LIN {X 0,Y 247.203,Z 467.136,A -85,B 0,C 180,E1 -18801.825,E2 -18801.825} C_VEL
LIN {X 0,Y 246.923,Z 469.012,A -85,B 0,C 180,E1 -18805.099,E2 -18805.099} C_VEL
LIN {X 0,Y 246.987,Z 469.369,A -85,B 0,C 180,E1 -18806.735,E2 -18806.735} C_VEL
LIN {X 0,Y 247.048,Z 469.339,A -85,B 0,C 180,E1 -18808.367,E2 -18808.367} C_VEL
LIN {X 0,Y 247.097,Z 468.891,A -85,B 0,C 180,E1 -18809.997,E2 -18809.997} C_VEL
LIN {X 0,Y 247.079,Z 468.012,A -85,B 0,C 180,E1 -18811.627,E2 -18811.627} C_VEL
LIN {X 0,Y 247.04,Z 466.727,A -85,B 0,C 180,E1 -18813.258,E2 -18813.258} C_VEL
LIN {X 0,Y 247.021,Z 464.571,A -85,B 0,C 180,E1 -18815.261,E2 -18815.261} C_VEL
LIN {X 0,Y 247.246,Z 460.184,A -85,B 0,C 180,E1 -18818.167,E2 -18818.167} C_VEL
LIN {X 0,Y 247.68,Z 455.238,A -85,B 0,C 180,E1 -18820.624,E2 -18820.624} C_VEL
LIN {X 0,Y 248.441,Z 448.994,A -85,B 0,C 180,E1 -18823.075,E2 -18823.075} C_VEL
LIN {X 0,Y 249.662,Z 441.211,A -85,B 0,C 180,E1 -18825.506,E2 -18825.506} C_VEL
LIN {X 0,Y 250.752,Z 434.213,A -85,B 0,C 180,E1 -18827.293,E2 -18827.293} C_VEL
LIN {X 0,Y 252.36,Z 424.659,A -85,B 0,C 180,E1 -18829.286,E2 -18829.286} C_VEL
LIN {X 0,Y 253.976,Z 413.923,A -85,B 0,C 180,E1 -18831.079,E2 -18831.079} C_VEL
LIN {X 0,Y 255.738,Z 402.097,A -85,B 0,C 180,E1 -18832.622,E2 -18832.622} C_VEL
LIN {X 0,Y 257.174,Z 390.548,A -85,B 0,C 180,E1 -18833.765,E2 -18833.765} C_VEL
LIN {X 0,Y 258.492,Z 377.529,A -85,B 0,C 180,E1 -18834.704,E2 -18834.704} C_VEL
LIN {X 0,Y 259.341,Z 364.879,A -85,B 0,C 180,E1 -18835.313,E2 -18835.313} C_VEL
LIN {X 0,Y 260.976,Z 308.011,A -85,B 0,C 180,E1 -18836.87,E2 -18836.87} C_VEL
LIN {X 0,Y 256.67,Z 271.586,A -85,B 0,C 180,E1 -18838.358,E2 -18838.358} C_VEL
LIN {X 0,Y 255.368,Z 263.288,A -85,B 0,C 180,E1 -18838.738,E2 -18838.738} C_VEL
LIN {X 0,Y 252.839,Z 256.196,A -85,B 0,C 180,E1 -18839.225,E2 -18839.225} C_VEL
LIN {X 0,Y 250.431,Z 244.513,A -85,B 0,C 180,E1 -18843.344,E2 -18843.344} C_VEL
LIN {X 0,Y 249.071,Z 238.465,A -85,B 0,C 180,E1 -18845.637,E2 -18845.637} C_VEL
LIN {X 0,Y 249.01,Z 238.469,A -85,B 0,C 180,E1 -18848.375,E2 -18848.375} C_VEL
LIN {X 0,Y 248.991,Z 238.469,A -85,B 0,C 180,E1 -18852.788,E2 -18852.788} C_VEL
LIN {X 0,Y 249.034,Z 238.465,A -85,B 0,C 180,E1 -18857.367,E2 -18857.367} C_VEL
LIN {X 0,Y 249.022,Z 238.468,A -85,B 0,C 180,E1 -18861.619,E2 -18861.619} C_VEL
LIN {X 0,Y 249.017,Z 238.467,A -85,B 0,C 180,E1 -18865.635,E2 -18865.635} C_VEL
LIN {X 0,Y 249.021,Z 238.466,A -85,B 0,C 180,E1 -18869.469,E2 -18869.469} C_VEL
LIN {X 0,Y 249.044,Z 238.463,A -85,B 0,C 180,E1 -18873.159,E2 -18873.159} C_VEL
LIN {X 0,Y 249.081,Z 238.456,A -85,B 0,C 180,E1 -18876.733,E2 -18876.733} C_VEL
LIN {X 0,Y 249.112,Z 238.452,A -85,B 0,C 180,E1 -18880.212,E2 -18880.212} C_VEL
LIN {X 0,Y 249.161,Z 238.449,A -85,B 0,C 180,E1 -18883.617,E2 -18883.617} C_VEL
LIN {X 0,Y 249.205,Z 238.44,A -85,B 0,C 180,E1 -18888.614,E2 -18888.614} C_VEL
LIN {X 0,Y 249.42,Z 238.411,A -85,B 0,C 180,E1 -18891.901,E2 -18891.901} C_VEL
LIN {X 0,Y 249.257,Z 238.437,A -85,B 0,C 180,E1 -18895.148,E2 -18895.148} C_VEL
LIN {X 0,Y 249.634,Z 238.385,A -85,B 0,C 180,E1 -18898.387,E2 -18898.387} C_VEL
LIN {X 0,Y 249.631,Z 238.366,A -85,B 0,C 180,E1 -18901.613,E2 -18901.613} C_VEL
LIN {X 0,Y 249.393,Z 238.414,A -85,B 0,C 180,E1 -18906.767,E2 -18906.767} C_VEL
LIN {X 0,Y 249.297,Z 238.427,A -85,B 0,C 180,E1 -18909.738,E2 -18909.738} C_VEL
LIN {X 0,Y 249.132,Z 238.432,A -85,B 0,C 180,E1 -18914.708,E2 -18914.708} C_VEL
LIN {X 0,Y 249.058,Z 238.455,A -85,B 0,C 180,E1 -18918.084,E2 -18918.084} C_VEL
LIN {X 0,Y 249.012,Z 238.464,A -85,B 0,C 180,E1 -18921.525,E2 -18921.525} C_VEL
LIN {X 0,Y 249.084,Z 238.456,A -85,B 0,C 180,E1 -18925.478,E2 -18925.478} C_VEL
LIN {X 0,Y 249.042,Z 238.46,A -85,B 0,C 180,E1 -18928.992,E2 -18928.992} C_VEL
LIN {X 0,Y 249.002,Z 238.469,A -85,B 0,C 180,E1 -18932.43,E2 -18932.43} C_VEL
LIN {X 0,Y 249.035,Z 238.465,A -85,B 0,C 180,E1 -18936.345,E2 -18936.345} C_VEL
LIN {X 0,Y 249.053,Z 238.461,A -85,B 0,C 180,E1 -18940.469,E2 -18940.469} C_VEL
LIN {X 0,Y 248.992,Z 238.457,A -85,B 0,C 180,E1 -18944.882,E2 -18944.882} C_VEL
LIN {X 0,Y 248.999,Z 238.46,A -85,B 0,C 180,E1 -18947.368,E2 -18947.368} C_VEL
LIN {X 0,Y 249.026,Z 238.457,A -85,B 0,C 180,E1 -18952.206,E2 -18952.206} C_VEL
LIN {X 0,Y 249.03,Z 238.464,A -85,B 0,C 180,E1 -18955.645,E2 -18955.645} C_VEL
LIN {X 0,Y 249.036,Z 238.464,A -85,B 0,C 180,E1 -18959.478,E2 -18959.478} C_VEL
LIN {X 0,Y 249.059,Z 238.459,A -85,B 0,C 180,E1 -18963.167,E2 -18963.167} C_VEL
LIN {X 0,Y 249.053,Z 238.458,A -85,B 0,C 180,E1 -18966.736,E2 -18966.736} C_VEL
LIN {X 0,Y 249.116,Z 238.454,A -85,B 0,C 180,E1 -18971.159,E2 -18971.159} C_VEL
LIN {X 0,Y 249.116,Z 238.559,A -85,B 0,C 180,E1 -18971.564,E2 -18971.564} C_VEL
LIN {X 0,Y 250.194,Z 241.443,A -85,B 0,C 180,E1 -18971.772,E2 -18971.772} C_VEL
LIN {X 0,Y 256.891,Z 255.902,A -85,B 0,C 180,E1 -18972.914,E2 -18972.914} C_VEL
LIN {X 0,Y 262.003,Z 270.873,A -85,B 0,C 180,E1 -18973.855,E2 -18973.855} C_VEL
LIN {X 0,Y 259.67,Z 343.56,A -85,B 0,C 180,E1 -18975.827,E2 -18975.827} C_VEL
LIN {X 0,Y 258.82,Z 356.25,A -85,B 0,C 180,E1 -18976.46,E2 -18976.46} C_VEL
LIN {X 0,Y 257.913,Z 367.725,A -85,B 0,C 180,E1 -18977.313,E2 -18977.313} C_VEL
LIN {X 0,Y 256.76,Z 380.047,A -85,B 0,C 180,E1 -18978.558,E2 -18978.558} C_VEL
LIN {X 0,Y 255.064,Z 391.695,A -85,B 0,C 180,E1 -18980.088,E2 -18980.088} C_VEL
LIN {X 0,Y 253.487,Z 402.134,A -85,B 0,C 180,E1 -18981.835,E2 -18981.835} C_VEL
LIN {X 0,Y 252.061,Z 410.678,A -85,B 0,C 180,E1 -18983.6,E2 -18983.6} C_VEL
LIN {X 0,Y 250.811,Z 418.54,A -85,B 0,C 180,E1 -18985.584,E2 -18985.584} C_VEL
LIN {X 0,Y 249.419,Z 426.253,A -85,B 0,C 180,E1 -18987.985,E2 -18987.985} C_VEL
LIN {X 0,Y 248.629,Z 431.513,A -85,B 0,C 180,E1 -18990.003,E2 -18990.003} C_VEL
LIN {X 0,Y 247.945,Z 436.619,A -85,B 0,C 180,E1 -18992.44,E2 -18992.44} C_VEL
LIN {X 0,Y 247.504,Z 440.592,A -85,B 0,C 180,E1 -18994.889,E2 -18994.889} C_VEL
LIN {X 0,Y 247.252,Z 442.647,A -85,B 0,C 180,E1 -18996.531,E2 -18996.531} C_VEL
LIN {X 0,Y 247.006,Z 444.293,A -85,B 0,C 180,E1 -18998.181,E2 -18998.181} C_VEL
LIN {X 0,Y 246.9,Z 445.534,A -85,B 0,C 180,E1 -18999.836,E2 -18999.836} C_VEL
LIN {X 0,Y 246.89,Z 446.331,A -85,B 0,C 180,E1 -19001.496,E2 -19001.496} C_VEL
LIN {X 0,Y 247.048,Z 446.719,A -85,B 0,C 180,E1 -19003.157,E2 -19003.157} C_VEL
LIN {X 0,Y 247.277,Z 446.714,A -85,B 0,C 180,E1 -19004.908,E2 -19004.908} C_VEL
LIN {X 0,Y 247.511,Z 446.329,A -85,B 0,C 180,E1 -19006.497,E2 -19006.497} C_VEL
LIN {X 0,Y 247.958,Z 445.48,A -85,B 0,C 180,E1 -19008.168,E2 -19008.168} C_VEL
LIN {X 0,Y 248.534,Z 444.221,A -85,B 0,C 180,E1 -19009.838,E2 -19009.838} C_VEL
LIN {X 0,Y 249.653,Z 441.509,A -85,B 0,C 180,E1 -19012.337,E2 -19012.337} C_VEL
LIN {X 0,Y 251.127,Z 437.727,A -85,B 0,C 180,E1 -19014.822,E2 -19014.822} C_VEL
LIN {X 0,Y 253.115,Z 432.322,A -85,B 0,C 180,E1 -19017.48,E2 -19017.48} C_VEL
LIN {X 0,Y 255.623,Z 425.225,A -85,B 0,C 180,E1 -19020.117,E2 -19020.117} C_VEL
LIN {X 0,Y 258.288,Z 417.007,A -85,B 0,C 180,E1 -19022.487,E2 -19022.487} C_VEL
LIN {X 0,Y 260.828,Z 408.416,A -85,B 0,C 180,E1 -19024.461,E2 -19024.461} C_VEL
LIN {X 0,Y 263.568,Z 398.096,A -85,B 0,C 180,E1 -19026.333,E2 -19026.333} C_VEL
LIN {X 0,Y 266.096,Z 387.21,A -85,B 0,C 180,E1 -19027.883,E2 -19027.883} C_VEL
LIN {X 0,Y 268.227,Z 375.469,A -85,B 0,C 180,E1 -19029.205,E2 -19029.205} C_VEL
LIN {X 0,Y 270.041,Z 363.177,A -85,B 0,C 180,E1 -19030.222,E2 -19030.222} C_VEL
LIN {X 0,Y 271.458,Z 349.994,A -85,B 0,C 180,E1 -19030.986,E2 -19030.986} C_VEL
LIN {X 0,Y 272.232,Z 337.682,A -85,B 0,C 180,E1 -19031.434,E2 -19031.434} C_VEL
LIN {X 0,Y 274.351,Z 284.179,A -85,B 0,C 180,E1 -19032.822,E2 -19032.822} C_VEL
LIN {X 0,Y 267.59,Z 269.785,A -85,B 0,C 180,E1 -19034.382,E2 -19034.382} C_VEL
LIN {X 0,Y 261.114,Z 257.839,A -85,B 0,C 180,E1 -19035.925,E2 -19035.925} C_VEL
LIN {X 0,Y 253.708,Z 246.432,A -85,B 0,C 180,E1 -19037.752,E2 -19037.752} C_VEL
LIN {X 0,Y 251.454,Z 242.928,A -85,B 0,C 180,E1 -19038.342,E2 -19038.342} C_VEL
LIN {X 0,Y 249.713,Z 240.612,A -85,B 0,C 180,E1 -19038.795,E2 -19038.795} C_VEL
LIN {X 0,Y 249.083,Z 238.458,A -85,B 0,C 180,E1 -19039.037,E2 -19039.037} C_VEL
LIN {X 0,Y 249.052,Z 238.46,A -85,B 0,C 180,E1 -19043.658,E2 -19043.658} C_VEL
LIN {X 0,Y 249.031,Z 238.463,A -85,B 0,C 180,E1 -19047.845,E2 -19047.845} C_VEL
LIN {X 0,Y 249.089,Z 238.456,A -85,B 0,C 180,E1 -19051.337,E2 -19051.337} C_VEL
LIN {X 0,Y 249.125,Z 238.452,A -85,B 0,C 180,E1 -19054.965,E2 -19054.965} C_VEL
LIN {X 0,Y 249.08,Z 238.458,A -85,B 0,C 180,E1 -19058.604,E2 -19058.604} C_VEL
LIN {X 0,Y 249.187,Z 238.438,A -85,B 0,C 180,E1 -19063.618,E2 -19063.618} C_VEL
LIN {X 0,Y 249.212,Z 238.432,A -85,B 0,C 180,E1 -19068.614,E2 -19068.614} C_VEL
LIN {X 0,Y 249.434,Z 238.413,A -85,B 0,C 180,E1 -19071.901,E2 -19071.901} C_VEL
LIN {X 0,Y 249.271,Z 238.431,A -85,B 0,C 180,E1 -19075.148,E2 -19075.148} C_VEL
LIN {X 0,Y 249.657,Z 238.373,A -85,B 0,C 180,E1 -19078.387,E2 -19078.387} C_VEL
LIN {X 0,Y 249.651,Z 238.383,A -85,B 0,C 180,E1 -19081.613,E2 -19081.613} C_VEL
LIN {X 0,Y 249.332,Z 238.415,A -85,B 0,C 180,E1 -19083.677,E2 -19083.677} C_VEL
LIN {X 0,Y 248.579,Z 238.52,A -85,B 0,C 180,E1 -19085.027,E2 -19085.027} C_VEL
LIN {X 0,Y 245.722,Z 238.875,A -85,B 0,C 180,E1 -19087.229,E2 -19087.229} C_VEL
LIN {X 0,Y 243.329,Z 239.172,A -85,B 0,C 180,E1 -19089.022,E2 -19089.022} C_VEL
LIN {X 0,Y 242.275,Z 239.305,A -85,B 0,C 180,E1 -19090.411,E2 -19090.411} C_VEL
LIN {X 0,Y 242.171,Z 239.31,A -85,B 0,C 180,E1 -19090.882,E2 -19090.882} C_VEL
LIN {X 0,Y 242.108,Z 239.325,A -85,B 0,C 180,E1 -19095.144,E2 -19095.144} C_VEL
LIN {X 0,Y 242.018,Z 239.335,A -85,B 0,C 180,E1 -19098.628,E2 -19098.628} C_VEL
LIN {X 0,Y 241.963,Z 239.336,A -85,B 0,C 180,E1 -19102.185,E2 -19102.185} C_VEL
LIN {X 0,Y 241.978,Z 239.332,A -85,B 0,C 180,E1 -19105.827,E2 -19105.827} C_VEL
LIN {X 0,Y 241.953,Z 239.336,A -85,B 0,C 180,E1 -19109.59,E2 -19109.59} C_VEL
LIN {X 0,Y 241.96,Z 239.335,A -85,B 0,C 180,E1 -19113.496,E2 -19113.496} C_VEL
LIN {X 0,Y 241.978,Z 239.314,A -85,B 0,C 180,E1 -19117.584,E2 -19117.584} C_VEL
LIN {X 0,Y 241.923,Z 239.349,A -85,B 0,C 180,E1 -19121.926,E2 -19121.926} C_VEL
LIN {X 0,Y 241.904,Z 239.396,A -85,B 0,C 180,E1 -19124.093,E2 -19124.093} C_VEL
LIN {X 0,Y 244.427,Z 247.713,A -85,B 0,C 180,E1 -19128.381,E2 -19128.381} C_VEL
LIN {X 0,Y 246.312,Z 254.372,A -85,B 0,C 180,E1 -19131.43,E2 -19131.43} C_VEL
LIN {X 0,Y 248.91,Z 258.983,A -85,B 0,C 180,E1 -19132.159,E2 -19132.159} C_VEL
LIN {X 0,Y 254.848,Z 270.286,A -85,B 0,C 180,E1 -19133.768,E2 -19133.768} C_VEL
LIN {X 0,Y 261.821,Z 284.82,A -85,B 0,C 180,E1 -19135.559,E2 -19135.559} C_VEL
LIN {X 0,Y 263.955,Z 290.021,A -85,B 0,C 180,E1 -19136.105,E2 -19136.105} C_VEL
LIN {X 0,Y 267.543,Z 313.214,A -85,B 0,C 180,E1 -19137.473,E2 -19137.473} C_VEL
LIN {X 0,Y 265.351,Z 364.24,A -85,B 0,C 180,E1 -19138.851,E2 -19138.851} C_VEL
LIN {X 0,Y 263.985,Z 377.838,A -85,B 0,C 180,E1 -19139.486,E2 -19139.486} C_VEL
LIN {X 0,Y 261.967,Z 390.55,A -85,B 0,C 180,E1 -19140.354,E2 -19140.354} C_VEL
LIN {X 0,Y 259.554,Z 402.464,A -85,B 0,C 180,E1 -19141.495,E2 -19141.495} C_VEL
LIN {X 0,Y 256.853,Z 413.883,A -85,B 0,C 180,E1 -19142.942,E2 -19142.942} C_VEL
LIN {X 0,Y 253.958,Z 424.203,A -85,B 0,C 180,E1 -19144.599,E2 -19144.599} C_VEL
LIN {X 0,Y 251.143,Z 433.502,A -85,B 0,C 180,E1 -19146.498,E2 -19146.498} C_VEL
LIN {X 0,Y 248.11,Z 442.53,A -85,B 0,C 180,E1 -19148.828,E2 -19148.828} C_VEL
LIN {X 0,Y 245.748,Z 449.9,A -85,B 0,C 180,E1 -19151.258,E2 -19151.258} C_VEL
LIN {X 0,Y 243.418,Z 456.556,A -85,B 0,C 180,E1 -19154.079,E2 -19154.079} C_VEL
LIN {X 0,Y 241.79,Z 461.028,A -85,B 0,C 180,E1 -19156.552,E2 -19156.552} C_VEL
LIN {X 0,Y 241.123,Z 463.407,A -85,B 0,C 180,E1 -19158.225,E2 -19158.225} C_VEL
LIN {X 0,Y 240.555,Z 465.363,A -85,B 0,C 180,E1 -19159.902,E2 -19159.902} C_VEL
LIN {X 0,Y 240.162,Z 466.905,A -85,B 0,C 180,E1 -19161.584,E2 -19161.584} C_VEL
LIN {X 0,Y 239.847,Z 468.719,A -85,B 0,C 180,E1 -19164.954,E2 -19164.954} C_VEL
LIN {X 0,Y 239.882,Z 469.052,A -85,B 0,C 180,E1 -19166.638,E2 -19166.638} C_VEL
LIN {X 0,Y 239.975,Z 468.998,A -85,B 0,C 180,E1 -19168.319,E2 -19168.319} C_VEL
LIN {X 0,Y 240.022,Z 468.506,A -85,B 0,C 180,E1 -19169.997,E2 -19169.997} C_VEL
LIN {X 0,Y 240.006,Z 467.602,A -85,B 0,C 180,E1 -19171.675,E2 -19171.675} C_VEL
LIN {X 0,Y 239.955,Z 466.293,A -85,B 0,C 180,E1 -19173.355,E2 -19173.355} C_VEL
LIN {X 0,Y 239.95,Z 464.329,A -85,B 0,C 180,E1 -19175.226,E2 -19175.226} C_VEL
LIN {X 0,Y 240.105,Z 461.075,A -85,B 0,C 180,E1 -19177.565,E2 -19177.565} C_VEL
LIN {X 0,Y 240.463,Z 456.468,A -85,B 0,C 180,E1 -19180.096,E2 -19180.096} C_VEL
LIN {X 0,Y 241.321,Z 449.467,A -85,B 0,C 180,E1 -19183.04,E2 -19183.04} C_VEL
LIN {X 0,Y 242.562,Z 441.881,A -85,B 0,C 180,E1 -19185.541,E2 -19185.541} C_VEL
LIN {X 0,Y 243.714,Z 434.867,A -85,B 0,C 180,E1 -19187.425,E2 -19187.425} C_VEL
LIN {X 0,Y 245.28,Z 425.71,A -85,B 0,C 180,E1 -19189.451,E2 -19189.451} C_VEL
LIN {X 0,Y 246.938,Z 415.436,A -85,B 0,C 180,E1 -19191.271,E2 -19191.271} C_VEL
LIN {X 0,Y 248.456,Z 405.625,A -85,B 0,C 180,E1 -19192.663,E2 -19192.663} C_VEL
LIN {X 0,Y 250.176,Z 393.195,A -85,B 0,C 180,E1 -19194.032,E2 -19194.032} C_VEL
LIN {X 0,Y 251.486,Z 381.401,A -85,B 0,C 180,E1 -19194.998,E2 -19194.998} C_VEL
LIN {X 0,Y 252.523,Z 368.688,A -85,B 0,C 180,E1 -19195.715,E2 -19195.715} C_VEL
LIN {X 0,Y 253.145,Z 352.376,A -85,B 0,C 180,E1 -19196.255,E2 -19196.255} C_VEL
LIN {X 0,Y 254.295,Z 307.444,A -85,B 0,C 180,E1 -19197.504,E2 -19197.504} C_VEL
LIN {X 0,Y 249.978,Z 270.919,A -85,B 0,C 180,E1 -19199.053,E2 -19199.053} C_VEL
LIN {X 0,Y 248.956,Z 265.195,A -85,B 0,C 180,E1 -19199.339,E2 -19199.339} C_VEL
LIN {X 0,Y 245.586,Z 255.846,A -85,B 0,C 180,E1 -19200.008,E2 -19200.008} C_VEL
LIN {X 0,Y 243.121,Z 244.14,A -85,B 0,C 180,E1 -19204.303,E2 -19204.303} C_VEL
LIN {X 0,Y 242.004,Z 239.343,A -85,B 0,C 180,E1 -19206.205,E2 -19206.205} C_VEL
LIN {X 0,Y 241.939,Z 239.35,A -85,B 0,C 180,E1 -19209.714,E2 -19209.714} C_VEL
LIN {X 0,Y 241.916,Z 239.351,A -85,B 0,C 180,E1 -19214.196,E2 -19214.196} C_VEL
LIN {X 0,Y 241.958,Z 239.347,A -85,B 0,C 180,E1 -19218.082,E2 -19218.082} C_VEL
LIN {X 0,Y 241.978,Z 239.342,A -85,B 0,C 180,E1 -19222.416,E2 -19222.416} C_VEL
LIN {X 0,Y 241.953,Z 239.344,A -85,B 0,C 180,E1 -19226.503,E2 -19226.503} C_VEL
LIN {X 0,Y 242.007,Z 239.338,A -85,B 0,C 180,E1 -19230.584,E2 -19230.584} C_VEL
LIN {X 0,Y 242.037,Z 239.334,A -85,B 0,C 180,E1 -19234.18,E2 -19234.18} C_VEL
LIN {X 0,Y 242.056,Z 239.331,A -85,B 0,C 180,E1 -19238.273,E2 -19238.273} C_VEL
LIN {X 0,Y 242.121,Z 239.326,A -85,B 0,C 180,E1 -19243.283,E2 -19243.283} C_VEL
LIN {X 0,Y 242.141,Z 239.32,A -85,B 0,C 180,E1 -19248.278,E2 -19248.278} C_VEL
LIN {X 0,Y 242.366,Z 239.29,A -85,B 0,C 180,E1 -19251.664,E2 -19251.664} C_VEL
LIN {X 0,Y 242.218,Z 239.313,A -85,B 0,C 180,E1 -19255.006,E2 -19255.006} C_VEL
LIN {X 0,Y 242.595,Z 239.261,A -85,B 0,C 180,E1 -19258.34,E2 -19258.34} C_VEL
LIN {X 0,Y 242.592,Z 239.241,A -85,B 0,C 180,E1 -19261.66,E2 -19261.66} C_VEL
LIN {X 0,Y 242.372,Z 239.29,A -85,B 0,C 180,E1 -19266.74,E2 -19266.74} C_VEL
LIN {X 0,Y 242.226,Z 239.308,A -85,B 0,C 180,E1 -19270.026,E2 -19270.026} C_VEL
LIN {X 0,Y 242.083,Z 239.311,A -85,B 0,C 180,E1 -19275.146,E2 -19275.146} C_VEL
LIN {X 0,Y 241.995,Z 239.338,A -85,B 0,C 180,E1 -19278.631,E2 -19278.631} C_VEL
LIN {X 0,Y 241.955,Z 239.344,A -85,B 0,C 180,E1 -19282.186,E2 -19282.186} C_VEL
LIN {X 0,Y 242.037,Z 239.334,A -85,B 0,C 180,E1 -19285.842,E2 -19285.842} C_VEL
LIN {X 0,Y 241.978,Z 239.338,A -85,B 0,C 180,E1 -19289.588,E2 -19289.588} C_VEL
LIN {X 0,Y 241.954,Z 239.342,A -85,B 0,C 180,E1 -19293.497,E2 -19293.497} C_VEL
LIN {X 0,Y 241.982,Z 239.341,A -85,B 0,C 180,E1 -19297.584,E2 -19297.584} C_VEL
LIN {X 0,Y 241.959,Z 239.344,A -85,B 0,C 180,E1 -19301.918,E2 -19301.918} C_VEL
LIN {X 0,Y 241.917,Z 239.336,A -85,B 0,C 180,E1 -19305.804,E2 -19305.804} C_VEL
LIN {X 0,Y 241.93,Z 239.347,A -85,B 0,C 180,E1 -19310.284,E2 -19310.284} C_VEL
LIN {X 0,Y 241.966,Z 239.342,A -85,B 0,C 180,E1 -19314.494,E2 -19314.494} C_VEL
LIN {X 0,Y 241.961,Z 239.345,A -85,B 0,C 180,E1 -19318.485,E2 -19318.485} C_VEL
LIN {X 0,Y 241.991,Z 239.341,A -85,B 0,C 180,E1 -19322.317,E2 -19322.317} C_VEL
LIN {X 0,Y 242.033,Z 239.335,A -85,B 0,C 180,E1 -19326.019,E2 -19326.019} C_VEL
LIN {X 0,Y 242.052,Z 239.333,A -85,B 0,C 180,E1 -19330.775,E2 -19330.775} C_VEL
LIN {X 0,Y 243.117,Z 242.269,A -85,B 0,C 180,E1 -19331.011,E2 -19331.011} C_VEL
LIN {X 0,Y 250.739,Z 258.529,A -85,B 0,C 180,E1 -19332.364,E2 -19332.364} C_VEL
LIN {X 0,Y 255.469,Z 272.48,A -85,B 0,C 180,E1 -19333.274,E2 -19333.274} C_VEL
LIN {X 0,Y 253.06,Z 343.957,A -85,B 0,C 180,E1 -19335.258,E2 -19335.258} C_VEL
LIN {X 0,Y 252.18,Z 356.417,A -85,B 0,C 180,E1 -19335.89,E2 -19335.89} C_VEL
LIN {X 0,Y 251.252,Z 367.929,A -85,B 0,C 180,E1 -19336.765,E2 -19336.765} C_VEL
LIN {X 0,Y 250.056,Z 380.285,A -85,B 0,C 180,E1 -19338.041,E2 -19338.041} C_VEL
LIN {X 0,Y 248.302,Z 391.953,A -85,B 0,C 180,E1 -19339.609,E2 -19339.609} C_VEL
LIN {X 0,Y 246.664,Z 402.405,A -85,B 0,C 180,E1 -19341.401,E2 -19341.401} C_VEL
LIN {X 0,Y 245.039,Z 411.836,A -85,B 0,C 180,E1 -19343.416,E2 -19343.416} C_VEL
LIN {X 0,Y 243.514,Z 420.897,A -85,B 0,C 180,E1 -19345.866,E2 -19345.866} C_VEL
LIN {X 0,Y 242.144,Z 428.227,A -85,B 0,C 180,E1 -19348.34,E2 -19348.34} C_VEL
LIN {X 0,Y 241.301,Z 434.084,A -85,B 0,C 180,E1 -19350.837,E2 -19350.837} C_VEL
LIN {X 0,Y 240.613,Z 438.721,A -85,B 0,C 180,E1 -19353.352,E2 -19353.352} C_VEL
LIN {X 0,Y 240.256,Z 442.364,A -85,B 0,C 180,E1 -19355.967,E2 -19355.967} C_VEL
LIN {X 0,Y 239.883,Z 444.8,A -85,B 0,C 180,E1 -19358.426,E2 -19358.426} C_VEL
LIN {X 0,Y 239.808,Z 445.979,A -85,B 0,C 180,E1 -19360.13,E2 -19360.13} C_VEL
LIN {X 0,Y 239.99,Z 447.071,A -85,B 0,C 180,E1 -19363.551,E2 -19363.551} C_VEL
LIN {X 0,Y 240.239,Z 447.035,A -85,B 0,C 180,E1 -19365.267,E2 -19365.267} C_VEL
LIN {X 0,Y 240.544,Z 446.572,A -85,B 0,C 180,E1 -19366.99,E2 -19366.99} C_VEL
LIN {X 0,Y 241.021,Z 445.678,A -85,B 0,C 180,E1 -19368.71,E2 -19368.71} C_VEL
LIN {X 0,Y 242.296,Z 442.972,A -85,B 0,C 180,E1 -19371.845,E2 -19371.845} C_VEL
LIN {X 0,Y 243.926,Z 439.154,A -85,B 0,C 180,E1 -19374.695,E2 -19374.695} C_VEL
LIN {X 0,Y 246.135,Z 433.406,A -85,B 0,C 180,E1 -19377.728,E2 -19377.728} C_VEL
LIN {X 0,Y 248.43,Z 427.372,A -85,B 0,C 180,E1 -19380.142,E2 -19380.142} C_VEL
LIN {X 0,Y 251.163,Z 419.752,A -85,B 0,C 180,E1 -19382.54,E2 -19382.54} C_VEL
LIN {X 0,Y 253.726,Z 411.531,A -85,B 0,C 180,E1 -19384.599,E2 -19384.599} C_VEL
LIN {X 0,Y 256.552,Z 401.625,A -85,B 0,C 180,E1 -19386.571,E2 -19386.571} C_VEL
LIN {X 0,Y 259.479,Z 390.344,A -85,B 0,C 180,E1 -19388.319,E2 -19388.319} C_VEL
LIN {X 0,Y 261.603,Z 379.544,A -85,B 0,C 180,E1 -19389.645,E2 -19389.645} C_VEL
LIN {X 0,Y 263.426,Z 368.513,A -85,B 0,C 180,E1 -19390.69,E2 -19390.69} C_VEL
LIN {X 0,Y 265.152,Z 355.149,A -85,B 0,C 180,E1 -19391.604,E2 -19391.604} C_VEL
LIN {X 0,Y 266.232,Z 341.893,A -85,B 0,C 180,E1 -19392.182,E2 -19392.182} C_VEL
LIN {X 0,Y 268.615,Z 286.422,A -85,B 0,C 180,E1 -19393.657,E2 -19393.657} C_VEL
LIN {X 0,Y 261.963,Z 272.273,A -85,B 0,C 180,E1 -19395.267,E2 -19395.267} C_VEL
LIN {X 0,Y 256.197,Z 261.74,A -85,B 0,C 180,E1 -19396.701,E2 -19396.701} C_VEL
LIN {X 0,Y 247.39,Z 248.085,A -85,B 0,C 180,E1 -19398.999,E2 -19398.999} C_VEL
LIN {X 0,Y 245.215,Z 244.854,A -85,B 0,C 180,E1 -19399.602,E2 -19399.602} C_VEL
LIN {X 0,Y 244.513,Z 243.904,A -85,B 0,C 180,E1 -19399.797,E2 -19399.797} C_VEL
LIN {X 0,Y 242.729,Z 241.705,A -85,B 0,C 180,E1 -19400.291,E2 -19400.291} C_VEL
LIN {X 0,Y 241.993,Z 239.339,A -85,B 0,C 180,E1 -19400.569,E2 -19400.569} C_VEL
LIN {X 0,Y 241.989,Z 239.342,A -85,B 0,C 180,E1 -19404.489,E2 -19404.489} C_VEL
LIN {X 0,Y 241.967,Z 239.338,A -85,B 0,C 180,E1 -19408.478,E2 -19408.478} C_VEL
LIN {X 0,Y 241.998,Z 239.331,A -85,B 0,C 180,E1 -19412.311,E2 -19412.311} C_VEL
LIN {X 0,Y 242.03,Z 239.327,A -85,B 0,C 180,E1 -19416.013,E2 -19416.013} C_VEL
LIN {X 0,Y 242.01,Z 239.331,A -85,B 0,C 180,E1 -19419.605,E2 -19419.605} C_VEL
LIN {X 0,Y 242.118,Z 239.322,A -85,B 0,C 180,E1 -19423.306,E2 -19423.306} C_VEL
LIN {X 0,Y 242.148,Z 239.314,A -85,B 0,C 180,E1 -19428.278,E2 -19428.278} C_VEL
LIN {X 0,Y 242.381,Z 239.293,A -85,B 0,C 180,E1 -19431.664,E2 -19431.664} C_VEL
LIN {X 0,Y 242.405,Z 239.279,A -85,B 0,C 180,E1 -19433.34,E2 -19433.34} C_VEL
LIN {X 0,Y 242.618,Z 239.25,A -85,B 0,C 180,E1 -19438.34,E2 -19438.34} C_VEL
LIN {X 0,Y 242.611,Z 239.259,A -85,B 0,C 180,E1 -19441.66,E2 -19441.66} C_VEL
LIN {X 0,Y 242.378,Z 239.285,A -85,B 0,C 180,E1 -19446.66,E2 -19446.66} C_VEL
LIN {X 0,Y 242.249,Z 239.308,A -85,B 0,C 180,E1 -19450.024,E2 -19450.024} C_VEL
LIN {X 0,Y 242.171,Z 239.31,A -85,B 0,C 180,E1 -19450.882,E2 -19450.882} C_VEL
LIN {X 0,Y 241.445,Z 239.4,A -85,B 0,C 180,E1 -19452.27,E2 -19452.27} C_VEL
LIN {X 0,Y 238.542,Z 239.77,A -85,B 0,C 180,E1 -19454.534,E2 -19454.534} C_VEL
LIN {X 0,Y 236.099,Z 240.067,A -85,B 0,C 180,E1 -19456.378,E2 -19456.378} C_VEL
LIN {X 0,Y 235.042,Z 240.198,A -85,B 0,C 180,E1 -19457.81,E2 -19457.81} C_VEL
LIN {X 0,Y 234.95,Z 240.209,A -85,B 0,C 180,E1 -19458.295,E2 -19458.295} C_VEL
LIN {X 0,Y 234.906,Z 240.22,A -85,B 0,C 180,E1 -19462.888,E2 -19462.888} C_VEL
LIN {X 0,Y 234.896,Z 240.217,A -85,B 0,C 180,E1 -19466.666,E2 -19466.666} C_VEL
LIN {X 0,Y 234.878,Z 240.219,A -85,B 0,C 180,E1 -19470.575,E2 -19470.575} C_VEL
LIN {X 0,Y 234.892,Z 240.221,A -85,B 0,C 180,E1 -19474.644,E2 -19474.644} C_VEL
LIN {X 0,Y 234.908,Z 240.191,A -85,B 0,C 180,E1 -19478.936,E2 -19478.936} C_VEL
LIN {X 0,Y 234.896,Z 240.384,A -85,B 0,C 180,E1 -19482.706,E2 -19482.706} C_VEL
LIN {X 0,Y 237.338,Z 248.366,A -85,B 0,C 180,E1 -19487.074,E2 -19487.074} C_VEL
LIN {X 0,Y 238.938,Z 253.915,A -85,B 0,C 180,E1 -19489.744,E2 -19489.744} C_VEL
LIN {X 0,Y 241.554,Z 258.478,A -85,B 0,C 180,E1 -19490.539,E2 -19490.539} C_VEL
LIN {X 0,Y 247.486,Z 269.065,A -85,B 0,C 180,E1 -19492.25,E2 -19492.25} C_VEL
LIN {X 0,Y 254.115,Z 282.629,A -85,B 0,C 180,E1 -19494.079,E2 -19494.079} C_VEL
LIN {X 0,Y 258.668,Z 293.05,A -85,B 0,C 180,E1 -19495.29,E2 -19495.29} C_VEL
LIN {X 0,Y 261.841,Z 314.42,A -85,B 0,C 180,E1 -19496.58,E2 -19496.58} C_VEL
LIN {X 0,Y 259.63,Z 363.67,A -85,B 0,C 180,E1 -19497.931,E2 -19497.931} C_VEL
LIN {X 0,Y 258.191,Z 377.418,A -85,B 0,C 180,E1 -19498.576,E2 -19498.576} C_VEL
LIN {X 0,Y 256.056,Z 390.472,A -85,B 0,C 180,E1 -19499.484,E2 -19499.484} C_VEL
LIN {X 0,Y 253.363,Z 403.104,A -85,B 0,C 180,E1 -19500.732,E2 -19500.732} C_VEL
LIN {X 0,Y 250.564,Z 414.341,A -85,B 0,C 180,E1 -19502.205,E2 -19502.205} C_VEL
LIN {X 0,Y 247.576,Z 424.508,A -85,B 0,C 180,E1 -19503.895,E2 -19503.895} C_VEL
LIN {X 0,Y 244.663,Z 433.669,A -85,B 0,C 180,E1 -19505.836,E2 -19505.836} C_VEL
LIN {X 0,Y 241.482,Z 442.613,A -85,B 0,C 180,E1 -19508.217,E2 -19508.217} C_VEL
LIN {X 0,Y 239.051,Z 449.872,A -85,B 0,C 180,E1 -19510.697,E2 -19510.697} C_VEL
LIN {X 0,Y 237.218,Z 454.746,A -85,B 0,C 180,E1 -19512.765,E2 -19512.765} C_VEL
LIN {X 0,Y 235.387,Z 459.538,A -85,B 0,C 180,E1 -19515.296,E2 -19515.296} C_VEL
LIN {X 0,Y 234.139,Z 463.24,A -85,B 0,C 180,E1 -19517.869,E2 -19517.869} C_VEL
LIN {X 0,Y 233.537,Z 465.17,A -85,B 0,C 180,E1 -19519.595,E2 -19519.595} C_VEL
LIN {X 0,Y 233.111,Z 466.664,A -85,B 0,C 180,E1 -19521.328,E2 -19521.328} C_VEL
LIN {X 0,Y 232.766,Z 468.427,A -85,B 0,C 180,E1 -19524.8,E2 -19524.8} C_VEL
LIN {X 0,Y 232.782,Z 468.736,A -85,B 0,C 180,E1 -19526.535,E2 -19526.535} C_VEL
LIN {X 0,Y 232.902,Z 468.646,A -85,B 0,C 180,E1 -19528.268,E2 -19528.268} C_VEL
LIN {X 0,Y 232.95,Z 468.119,A -85,B 0,C 180,E1 -19529.997,E2 -19529.997} C_VEL
LIN {X 0,Y 232.934,Z 467.192,A -85,B 0,C 180,E1 -19531.726,E2 -19531.726} C_VEL
LIN {X 0,Y 232.852,Z 465.855,A -85,B 0,C 180,E1 -19533.457,E2 -19533.457} C_VEL
LIN {X 0,Y 232.897,Z 463.005,A -85,B 0,C 180,E1 -19536.059,E2 -19536.059} C_VEL
LIN {X 0,Y 233.121,Z 459.099,A -85,B 0,C 180,E1 -19538.665,E2 -19538.665} C_VEL
LIN {X 0,Y 233.618,Z 454.033,A -85,B 0,C 180,E1 -19541.272,E2 -19541.272} C_VEL
LIN {X 0,Y 234.586,Z 447.662,A -85,B 0,C 180,E1 -19543.863,E2 -19543.863} C_VEL
LIN {X 0,Y 235.928,Z 439.657,A -85,B 0,C 180,E1 -19546.434,E2 -19546.434} C_VEL
LIN {X 0,Y 237.295,Z 431.3,A -85,B 0,C 180,E1 -19548.603,E2 -19548.603} C_VEL
LIN {X 0,Y 239.076,Z 421.504,A -85,B 0,C 180,E1 -19550.651,E2 -19550.651} C_VEL
LIN {X 0,Y 240.889,Z 410.286,A -85,B 0,C 180,E1 -19552.509,E2 -19552.509} C_VEL
LIN {X 0,Y 242.676,Z 399.311,A -85,B 0,C 180,E1 -19553.913,E2 -19553.913} C_VEL
LIN {X 0,Y 244.199,Z 387.142,A -85,B 0,C 180,E1 -19555.113,E2 -19555.113} C_VEL
LIN {X 0,Y 245.432,Z 374.604,A -85,B 0,C 180,E1 -19556.001,E2 -19556.001} C_VEL
LIN {X 0,Y 246.326,Z 361.542,A -85,B 0,C 180,E1 -19556.583,E2 -19556.583} C_VEL
LIN {X 0,Y 247.777,Z 308.364,A -85,B 0,C 180,E1 -19558.112,E2 -19558.112} C_VEL
LIN {X 0,Y 243.665,Z 272.715,A -85,B 0,C 180,E1 -19559.67,E2 -19559.67} C_VEL
LIN {X 0,Y 242.696,Z 267.43,A -85,B 0,C 180,E1 -19559.947,E2 -19559.947} C_VEL
LIN {X 0,Y 238.265,Z 255.416,A -85,B 0,C 180,E1 -19560.878,E2 -19560.878} C_VEL
LIN {X 0,Y 235.979,Z 244.696,A -85,B 0,C 180,E1 -19564.963,E2 -19564.963} C_VEL
LIN {X 0,Y 234.964,Z 240.22,A -85,B 0,C 180,E1 -19566.801,E2 -19566.801} C_VEL
LIN {X 0,Y 234.865,Z 240.229,A -85,B 0,C 180,E1 -19571.163,E2 -19571.163} C_VEL
LIN {X 0,Y 234.913,Z 240.224,A -85,B 0,C 180,E1 -19575.881,E2 -19575.881} C_VEL
LIN {X 0,Y 234.919,Z 240.223,A -85,B 0,C 180,E1 -19578.84,E2 -19578.84} C_VEL
LIN {X 0,Y 234.931,Z 240.221,A -85,B 0,C 180,E1 -19581.081,E2 -19581.081} C_VEL
LIN {X 0,Y 234.907,Z 240.226,A -85,B 0,C 180,E1 -19585.358,E2 -19585.358} C_VEL
LIN {X 0,Y 234.902,Z 240.225,A -85,B 0,C 180,E1 -19589.428,E2 -19589.428} C_VEL
LIN {X 0,Y 234.964,Z 240.217,A -85,B 0,C 180,E1 -19593.79,E2 -19593.79} C_VEL
LIN {X 0,Y 235.016,Z 240.209,A -85,B 0,C 180,E1 -19598.97,E2 -19598.97} C_VEL
LIN {X 0,Y 235.057,Z 240.204,A -85,B 0,C 180,E1 -19603.062,E2 -19603.062} C_VEL
LIN {X 0,Y 235.073,Z 240.2,A -85,B 0,C 180,E1 -19607.92,E2 -19607.92} C_VEL
LIN {X 0,Y 235.296,Z 240.172,A -85,B 0,C 180,E1 -19611.411,E2 -19611.411} C_VEL
LIN {X 0,Y 235.338,Z 240.166,A -85,B 0,C 180,E1 -19613.14,E2 -19613.14} C_VEL
LIN {X 0,Y 235.555,Z 240.138,A -85,B 0,C 180,E1 -19618.29,E2 -19618.29} C_VEL
LIN {X 0,Y 235.552,Z 240.116,A -85,B 0,C 180,E1 -19621.71,E2 -19621.71} C_VEL
LIN {X 0,Y 235.329,Z 240.169,A -85,B 0,C 180,E1 -19626.861,E2 -19626.861} C_VEL
LIN {X 0,Y 235.174,Z 240.187,A -85,B 0,C 180,E1 -19630.33,E2 -19630.33} C_VEL
LIN {X 0,Y 235.034,Z 240.191,A -85,B 0,C 180,E1 -19635.612,E2 -19635.612} C_VEL
LIN {X 0,Y 234.934,Z 240.219,A -85,B 0,C 180,E1 -19639.212,E2 -19639.212} C_VEL
LIN {X 0,Y 234.91,Z 240.219,A -85,B 0,C 180,E1 -19642.888,E2 -19642.888} C_VEL
LIN {X 0,Y 234.937,Z 240.221,A -85,B 0,C 180,E1 -19646.662,E2 -19646.662} C_VEL
LIN {X 0,Y 234.893,Z 240.226,A -85,B 0,C 180,E1 -19650.574,E2 -19650.574} C_VEL
LIN {X 0,Y 234.908,Z 240.221,A -85,B 0,C 180,E1 -19654.642,E2 -19654.642} C_VEL
LIN {X 0,Y 234.944,Z 240.213,A -85,B 0,C 180,E1 -19658.957,E2 -19658.957} C_VEL
LIN {X 0,Y 234.939,Z 240.215,A -85,B 0,C 180,E1 -19663.474,E2 -19663.474} C_VEL
LIN {X 0,Y 234.859,Z 240.227,A -85,B 0,C 180,E1 -19668.427,E2 -19668.427} C_VEL
LIN {X 0,Y 234.901,Z 240.219,A -85,B 0,C 180,E1 -19671.084,E2 -19671.084} C_VEL
LIN {X 0,Y 234.913,Z 240.221,A -85,B 0,C 180,E1 -19675.367,E2 -19675.367} C_VEL
LIN {X 0,Y 234.911,Z 240.223,A -85,B 0,C 180,E1 -19679.436,E2 -19679.436} C_VEL
LIN {X 0,Y 234.985,Z 240.215,A -85,B 0,C 180,E1 -19683.799,E2 -19683.799} C_VEL
LIN {X 0,Y 234.983,Z 240.212,A -85,B 0,C 180,E1 -19688.973,E2 -19688.973} C_VEL
LIN {X 0,Y 234.986,Z 240.213,A -85,B 0,C 180,E1 -19689.95,E2 -19689.95} C_VEL
LIN {X 0,Y 236.08,Z 243.179,A -85,B 0,C 180,E1 -19690.207,E2 -19690.207} C_VEL
LIN {X 0,Y 244.604,Z 261.036,A -85,B 0,C 180,E1 -19691.782,E2 -19691.782} C_VEL
LIN {X 0,Y 248.931,Z 273.821,A -85,B 0,C 180,E1 -19692.651,E2 -19692.651} C_VEL
LIN {X 0,Y 246.529,Z 343.552,A -85,B 0,C 180,E1 -19694.624,E2 -19694.624} C_VEL
LIN {X 0,Y 245.59,Z 356.571,A -85,B 0,C 180,E1 -19695.292,E2 -19695.292} C_VEL
LIN {X 0,Y 244.619,Z 368.129,A -85,B 0,C 180,E1 -19696.188,E2 -19696.188} C_VEL
LIN {X 0,Y 243.374,Z 380.515,A -85,B 0,C 180,E1 -19697.496,E2 -19697.496} C_VEL
LIN {X 0,Y 241.557,Z 392.204,A -85,B 0,C 180,E1 -19699.103,E2 -19699.103} C_VEL
LIN {X 0,Y 239.855,Z 402.669,A -85,B 0,C 180,E1 -19700.943,E2 -19700.943} C_VEL
LIN {X 0,Y 238.289,Z 411.238,A -85,B 0,C 180,E1 -19702.803,E2 -19702.803} C_VEL
LIN {X 0,Y 236.927,Z 419.117,A -85,B 0,C 180,E1 -19704.898,E2 -19704.898} C_VEL
LIN {X 0,Y 235.448,Z 426.848,A -85,B 0,C 180,E1 -19707.437,E2 -19707.437} C_VEL
LIN {X 0,Y 234.469,Z 433.027,A -85,B 0,C 180,E1 -19710.003,E2 -19710.003} C_VEL
LIN {X 0,Y 233.686,Z 437.955,A -85,B 0,C 180,E1 -19712.589,E2 -19712.589} C_VEL
LIN {X 0,Y 233.271,Z 441.758,A -85,B 0,C 180,E1 -19715.188,E2 -19715.188} C_VEL
LIN {X 0,Y 232.996,Z 443.735,A -85,B 0,C 180,E1 -19716.932,E2 -19716.932} C_VEL
LIN {X 0,Y 232.785,Z 445.299,A -85,B 0,C 180,E1 -19718.685,E2 -19718.685} C_VEL
LIN {X 0,Y 232.714,Z 446.405,A -85,B 0,C 180,E1 -19720.442,E2 -19720.442} C_VEL
LIN {X 0,Y 232.774,Z 447.108,A -85,B 0,C 180,E1 -19722.203,E2 -19722.203} C_VEL
LIN {X 0,Y 233.168,Z 447.381,A -85,B 0,C 180,E1 -19725.306,E2 -19725.306} C_VEL
LIN {X 0,Y 233.583,Z 446.809,A -85,B 0,C 180,E1 -19727.512,E2 -19727.512} C_VEL
LIN {X 0,Y 234.11,Z 445.877,A -85,B 0,C 180,E1 -19729.284,E2 -19729.284} C_VEL
LIN {X 0,Y 235.372,Z 443.368,A -85,B 0,C 180,E1 -19732.235,E2 -19732.235} C_VEL
LIN {X 0,Y 237.275,Z 439.145,A -85,B 0,C 180,E1 -19735.436,E2 -19735.436} C_VEL
LIN {X 0,Y 239.452,Z 433.833,A -85,B 0,C 180,E1 -19738.295,E2 -19738.295} C_VEL
LIN {X 0,Y 242.128,Z 427.164,A -85,B 0,C 180,E1 -19741.012,E2 -19741.012} C_VEL
LIN {X 0,Y 244.558,Z 420.667,A -85,B 0,C 180,E1 -19743.094,E2 -19743.094} C_VEL
LIN {X 0,Y 247.169,Z 412.803,A -85,B 0,C 180,E1 -19745.155,E2 -19745.155} C_VEL
LIN {X 0,Y 250.101,Z 403.116,A -85,B 0,C 180,E1 -19747.168,E2 -19747.168} C_VEL
LIN {X 0,Y 253.14,Z 391.951,A -85,B 0,C 180,E1 -19748.979,E2 -19748.979} C_VEL
LIN {X 0,Y 255.336,Z 381.745,A -85,B 0,C 180,E1 -19750.302,E2 -19750.302} C_VEL
LIN {X 0,Y 257.371,Z 370.162,A -85,B 0,C 180,E1 -19751.466,E2 -19751.466} C_VEL
LIN {X 0,Y 259.222,Z 356.993,A -85,B 0,C 180,E1 -19752.407,E2 -19752.407} C_VEL
LIN {X 0,Y 260.397,Z 344.025,A -85,B 0,C 180,E1 -19753.03,E2 -19753.03} C_VEL
LIN {X 0,Y 262.934,Z 288.643,A -85,B 0,C 180,E1 -19754.532,E2 -19754.532} C_VEL
LIN {X 0,Y 256.067,Z 274.215,A -85,B 0,C 180,E1 -19756.273,E2 -19756.273} C_VEL
LIN {X 0,Y 251.525,Z 265.958,A -85,B 0,C 180,E1 -19757.459,E2 -19757.459} C_VEL
LIN {X 0,Y 243.298,Z 253.182,A -85,B 0,C 180,E1 -19759.696,E2 -19759.696} C_VEL
LIN {X 0,Y 240.291,Z 248.885,A -85,B 0,C 180,E1 -19760.563,E2 -19760.563} C_VEL
LIN {X 0,Y 238.08,Z 245.391,A -85,B 0,C 180,E1 -19761.236,E2 -19761.236} C_VEL
LIN {X 0,Y 235.759,Z 242.674,A -85,B 0,C 180,E1 -19761.924,E2 -19761.924} C_VEL
LIN {X 0,Y 234.972,Z 240.21,A -85,B 0,C 180,E1 -19762.249,E2 -19762.249} C_VEL
LIN {X 0,Y 234.95,Z 240.22,A -85,B 0,C 180,E1 -19767.423,E2 -19767.423} C_VEL
LIN {X 0,Y 234.943,Z 240.216,A -85,B 0,C 180,E1 -19771.405,E2 -19771.405} C_VEL
LIN {X 0,Y 234.969,Z 240.212,A -85,B 0,C 180,E1 -19775.244,E2 -19775.244} C_VEL
LIN {X 0,Y 234.98,Z 240.213,A -85,B 0,C 180,E1 -19778.967,E2 -19778.967} C_VEL
LIN {X 0,Y 235.055,Z 240.204,A -85,B 0,C 180,E1 -19783.086,E2 -19783.086} C_VEL
LIN {X 0,Y 235.083,Z 240.197,A -85,B 0,C 180,E1 -19787.92,E2 -19787.92} C_VEL
LIN {X 0,Y 235.31,Z 240.176,A -85,B 0,C 180,E1 -19791.411,E2 -19791.411} C_VEL
LIN {X 0,Y 235.355,Z 240.158,A -85,B 0,C 180,E1 -19793.14,E2 -19793.14} C_VEL
LIN {X 0,Y 235.578,Z 240.127,A -85,B 0,C 180,E1 -19798.29,E2 -19798.29} C_VEL
LIN {X 0,Y 235.57,Z 240.136,A -85,B 0,C 180,E1 -19801.709,E2 -19801.709} C_VEL
LIN {X 0,Y 235.329,Z 240.161,A -85,B 0,C 180,E1 -19806.861,E2 -19806.861} C_VEL
LIN {X 0,Y 235.174,Z 240.19,A -85,B 0,C 180,E1 -19810.329,E2 -19810.329} C_VEL
LIN {X 0,Y 235.059,Z 240.201,A -85,B 0,C 180,E1 -19815.61,E2 -19815.61} C_VEL
LIN {X 0,Y 234.95,Z 240.209,A -85,B 0,C 180,E1 -19818.295,E2 -19818.295} C_VEL
LIN {X 0,Y 234.263,Z 240.303,A -85,B 0,C 180,E1 -19819.726,E2 -19819.726} C_VEL
LIN {X 0,Y 231.401,Z 240.656,A -85,B 0,C 180,E1 -19822.059,E2 -19822.059} C_VEL
LIN {X 0,Y 228.978,Z 240.963,A -85,B 0,C 180,E1 -19823.962,E2 -19823.962} C_VEL
LIN {X 0,Y 227.939,Z 241.081,A -85,B 0,C 180,E1 -19825.439,E2 -19825.439} C_VEL
LIN {X 0,Y 227.854,Z 241.091,A -85,B 0,C 180,E1 -19825.939,E2 -19825.939} C_VEL
LIN {X 0,Y 227.858,Z 241.092,A -85,B 0,C 180,E1 -19830.277,E2 -19830.277} C_VEL
LIN {X 0,Y 227.862,Z 241.091,A -85,B 0,C 180,E1 -19833.723,E2 -19833.723} C_VEL
LIN {X 0,Y 227.836,Z 241.072,A -85,B 0,C 180,E1 -19838.093,E2 -19838.093} C_VEL
LIN {X 0,Y 227.83,Z 241.166,A -85,B 0,C 180,E1 -19841.06,E2 -19841.06} C_VEL
LIN {X 0,Y 230.346,Z 249.387,A -85,B 0,C 180,E1 -19845.847,E2 -19845.847} C_VEL
LIN {X 0,Y 231.518,Z 253.355,A -85,B 0,C 180,E1 -19847.875,E2 -19847.875} C_VEL
LIN {X 0,Y 234.222,Z 257.957,A -85,B 0,C 180,E1 -19848.767,E2 -19848.767} C_VEL
LIN {X 0,Y 240.63,Z 268.975,A -85,B 0,C 180,E1 -19850.757,E2 -19850.757} C_VEL
LIN {X 0,Y 247.46,Z 282.473,A -85,B 0,C 180,E1 -19852.76,E2 -19852.76} C_VEL
LIN {X 0,Y 253.288,Z 295.517,A -85,B 0,C 180,E1 -19854.392,E2 -19854.392} C_VEL
LIN {X 0,Y 256.212,Z 315.565,A -85,B 0,C 180,E1 -19855.646,E2 -19855.646} C_VEL
LIN {X 0,Y 253.921,Z 363.88,A -85,B 0,C 180,E1 -19856.999,E2 -19856.999} C_VEL
LIN {X 0,Y 252.425,Z 377.461,A -85,B 0,C 180,E1 -19857.653,E2 -19857.653} C_VEL
LIN {X 0,Y 250.215,Z 390.414,A -85,B 0,C 180,E1 -19858.575,E2 -19858.575} C_VEL
LIN {X 0,Y 247.633,Z 402.191,A -85,B 0,C 180,E1 -19859.751,E2 -19859.751} C_VEL
LIN {X 0,Y 244.703,Z 413.537,A -85,B 0,C 180,E1 -19861.244,E2 -19861.244} C_VEL
LIN {X 0,Y 241.569,Z 423.798,A -85,B 0,C 180,E1 -19862.961,E2 -19862.961} C_VEL
LIN {X 0,Y 238.217,Z 433.846,A -85,B 0,C 180,E1 -19865.139,E2 -19865.139} C_VEL
LIN {X 0,Y 234.887,Z 442.703,A -85,B 0,C 180,E1 -19867.573,E2 -19867.573} C_VEL
LIN {X 0,Y 232.446,Z 449.589,A -85,B 0,C 180,E1 -19870.004,E2 -19870.004} C_VEL
LIN {X 0,Y 230.409,Z 454.693,A -85,B 0,C 180,E1 -19872.239,E2 -19872.239} C_VEL
LIN {X 0,Y 228.512,Z 459.426,A -85,B 0,C 180,E1 -19874.844,E2 -19874.844} C_VEL
LIN {X 0,Y 227.147,Z 463.072,A -85,B 0,C 180,E1 -19877.489,E2 -19877.489} C_VEL
LIN {X 0,Y 226.535,Z 464.974,A -85,B 0,C 180,E1 -19879.27,E2 -19879.27} C_VEL
LIN {X 0,Y 225.77,Z 467.468,A -85,B 0,C 180,E1 -19882.845,E2 -19882.845} C_VEL
LIN {X 0,Y 225.689,Z 468.28,A -85,B 0,C 180,E1 -19885.196,E2 -19885.196} C_VEL
LIN {X 0,Y 225.829,Z 468.284,A -85,B 0,C 180,E1 -19888.213,E2 -19888.213} C_VEL
LIN {X 0,Y 225.88,Z 467.732,A -85,B 0,C 180,E1 -19889.997,E2 -19889.997} C_VEL
LIN {X 0,Y 225.862,Z 466.78,A -85,B 0,C 180,E1 -19891.78,E2 -19891.78} C_VEL
LIN {X 0,Y 225.741,Z 464.038,A -85,B 0,C 180,E1 -19894.959,E2 -19894.959} C_VEL
LIN {X 0,Y 225.966,Z 459.997,A -85,B 0,C 180,E1 -19898.041,E2 -19898.041} C_VEL
LIN {X 0,Y 226.406,Z 455.265,A -85,B 0,C 180,E1 -19900.73,E2 -19900.73} C_VEL
LIN {X 0,Y 227.237,Z 449.256,A -85,B 0,C 180,E1 -19903.408,E2 -19903.408} C_VEL
LIN {X 0,Y 228.525,Z 441.76,A -85,B 0,C 180,E1 -19906.063,E2 -19906.063} C_VEL
LIN {X 0,Y 229.808,Z 434.577,A -85,B 0,C 180,E1 -19908.131,E2 -19908.131} C_VEL
LIN {X 0,Y 231.652,Z 424.833,A -85,B 0,C 180,E1 -19910.414,E2 -19910.414} C_VEL
LIN {X 0,Y 233.412,Z 414.485,A -85,B 0,C 180,E1 -19912.336,E2 -19912.336} C_VEL
LIN {X 0,Y 235.319,Z 403.014,A -85,B 0,C 180,E1 -19914.006,E2 -19914.006} C_VEL
LIN {X 0,Y 237.023,Z 391.073,A -85,B 0,C 180,E1 -19915.34,E2 -19915.34} C_VEL
LIN {X 0,Y 238.422,Z 378.6,A -85,B 0,C 180,E1 -19916.353,E2 -19916.353} C_VEL
LIN {X 0,Y 239.569,Z 364.707,A -85,B 0,C 180,E1 -19917.099,E2 -19917.099} C_VEL
LIN {X 0,Y 241.381,Z 310.175,A -85,B 0,C 180,E1 -19918.713,E2 -19918.713} C_VEL
LIN {X 0,Y 237.32,Z 274.173,A -85,B 0,C 180,E1 -19920.336,E2 -19920.336} C_VEL
LIN {X 0,Y 236.345,Z 269.307,A -85,B 0,C 180,E1 -19920.611,E2 -19920.611} C_VEL
LIN {X 0,Y 230.991,Z 255.087,A -85,B 0,C 180,E1 -19921.763,E2 -19921.763} C_VEL
LIN {X 0,Y 229.099,Z 246.274,A -85,B 0,C 180,E1 -19925.25,E2 -19925.25} C_VEL
LIN {X 0,Y 227.925,Z 241.096,A -85,B 0,C 180,E1 -19927.405,E2 -19927.405} C_VEL
LIN {X 0,Y 227.793,Z 241.11,A -85,B 0,C 180,E1 -19932.737,E2 -19932.737} C_VEL
LIN {X 0,Y 227.884,Z 241.099,A -85,B 0,C 180,E1 -19937.275,E2 -19937.275} C_VEL
LIN {X 0,Y 227.843,Z 241.106,A -85,B 0,C 180,E1 -19941.909,E2 -19941.909} C_VEL
LIN {X 0,Y 227.853,Z 241.101,A -85,B 0,C 180,E1 -19946.373,E2 -19946.373} C_VEL
LIN {X 0,Y 227.89,Z 241.097,A -85,B 0,C 180,E1 -19950.434,E2 -19950.434} C_VEL
LIN {X 0,Y 227.903,Z 241.095,A -85,B 0,C 180,E1 -19954.423,E2 -19954.423} C_VEL
LIN {X 0,Y 227.978,Z 241.085,A -85,B 0,C 180,E1 -19958.289,E2 -19958.289} C_VEL
LIN {X 0,Y 227.999,Z 241.082,A -85,B 0,C 180,E1 -19962.826,E2 -19962.826} C_VEL
LIN {X 0,Y 228.03,Z 241.078,A -85,B 0,C 180,E1 -19967.541,E2 -19967.541} C_VEL
LIN {X 0,Y 228.233,Z 241.054,A -85,B 0,C 180,E1 -19971.143,E2 -19971.143} C_VEL
LIN {X 0,Y 228.289,Z 241.043,A -85,B 0,C 180,E1 -19972.927,E2 -19972.927} C_VEL
LIN {X 0,Y 228.514,Z 241.015,A -85,B 0,C 180,E1 -19978.238,E2 -19978.238} C_VEL
LIN {X 0,Y 228.511,Z 240.992,A -85,B 0,C 180,E1 -19981.763,E2 -19981.763} C_VEL
LIN {X 0,Y 228.279,Z 241.049,A -85,B 0,C 180,E1 -19987.074,E2 -19987.074} C_VEL
LIN {X 0,Y 228.105,Z 241.066,A -85,B 0,C 180,E1 -19990.653,E2 -19990.653} C_VEL
LIN {X 0,Y 227.982,Z 241.069,A -85,B 0,C 180,E1 -19996.108,E2 -19996.108} C_VEL
LIN {X 0,Y 227.885,Z 241.096,A -85,B 0,C 180,E1 -20001.721,E2 -20001.721} C_VEL
LIN {X 0,Y 227.912,Z 241.096,A -85,B 0,C 180,E1 -20006.605,E2 -20006.605} C_VEL
LIN {X 0,Y 227.868,Z 241.098,A -85,B 0,C 180,E1 -20010.294,E2 -20010.294} C_VEL
LIN {X 0,Y 227.852,Z 241.099,A -85,B 0,C 180,E1 -20013.725,E2 -20013.725} C_VEL
LIN {X 0,Y 227.845,Z 241.103,A -85,B 0,C 180,E1 -20018.091,E2 -20018.091} C_VEL
LIN {X 0,Y 227.885,Z 241.094,A -85,B 0,C 180,E1 -20022.726,E2 -20022.726} C_VEL
LIN {X 0,Y 227.792,Z 241.1,A -85,B 0,C 180,E1 -20027.263,E2 -20027.263} C_VEL
LIN {X 0,Y 227.827,Z 241.097,A -85,B 0,C 180,E1 -20031.914,E2 -20031.914} C_VEL
LIN {X 0,Y 227.866,Z 241.1,A -85,B 0,C 180,E1 -20036.383,E2 -20036.383} C_VEL
LIN {X 0,Y 227.894,Z 241.098,A -85,B 0,C 180,E1 -20040.441,E2 -20040.441} C_VEL
LIN {X 0,Y 227.917,Z 241.092,A -85,B 0,C 180,E1 -20044.431,E2 -20044.431} C_VEL
LIN {X 0,Y 227.942,Z 241.089,A -85,B 0,C 180,E1 -20049.086,E2 -20049.086} C_VEL
LIN {X 0,Y 228.931,Z 243.913,A -85,B 0,C 180,E1 -20049.329,E2 -20049.329} C_VEL
LIN {X 0,Y 237.03,Z 260.509,A -85,B 0,C 180,E1 -20050.901,E2 -20050.901} C_VEL
LIN {X 0,Y 240.325,Z 268.752,A -85,B 0,C 180,E1 -20051.553,E2 -20051.553} C_VEL
LIN {X 0,Y 242.296,Z 274.673,A -85,B 0,C 180,E1 -20051.965,E2 -20051.965} C_VEL
LIN {X 0,Y 239.96,Z 344.43,A -85,B 0,C 180,E1 -20054.014,E2 -20054.014} C_VEL
LIN {X 0,Y 239.018,Z 356.731,A -85,B 0,C 180,E1 -20054.66,E2 -20054.66} C_VEL
LIN {X 0,Y 238.016,Z 368.327,A -85,B 0,C 180,E1 -20055.578,E2 -20055.578} C_VEL
LIN {X 0,Y 236.714,Z 380.745,A -85,B 0,C 180,E1 -20056.92,E2 -20056.92} C_VEL
LIN {X 0,Y 234.833,Z 392.455,A -85,B 0,C 180,E1 -20058.569,E2 -20058.569} C_VEL
LIN {X 0,Y 233.062,Z 402.933,A -85,B 0,C 180,E1 -20060.457,E2 -20060.457} C_VEL
LIN {X 0,Y 231.273,Z 412.394,A -85,B 0,C 180,E1 -20062.584,E2 -20062.584} C_VEL
LIN {X 0,Y 229.63,Z 421.472,A -85,B 0,C 180,E1 -20065.176,E2 -20065.176} C_VEL
LIN {X 0,Y 228.163,Z 428.814,A -85,B 0,C 180,E1 -20067.797,E2 -20067.797} C_VEL
LIN {X 0,Y 227.086,Z 435.535,A -85,B 0,C 180,E1 -20070.89,E2 -20070.89} C_VEL
LIN {X 0,Y 226.427,Z 439.985,A -85,B 0,C 180,E1 -20073.562,E2 -20073.562} C_VEL
LIN {X 0,Y 226.107,Z 443.025,A -85,B 0,C 180,E1 -20075.927,E2 -20075.927} C_VEL
LIN {X 0,Y 225.672,Z 445.776,A -85,B 0,C 180,E1 -20078.961,E2 -20078.961} C_VEL
LIN {X 0,Y 225.705,Z 447.498,A -85,B 0,C 180,E1 -20082.592,E2 -20082.592} C_VEL
LIN {X 0,Y 226.104,Z 447.716,A -85,B 0,C 180,E1 -20085.51,E2 -20085.51} C_VEL
LIN {X 0,Y 226.632,Z 447.046,A -85,B 0,C 180,E1 -20088.067,E2 -20088.067} C_VEL
LIN {X 0,Y 227.219,Z 446.075,A -85,B 0,C 180,E1 -20089.893,E2 -20089.893} C_VEL
LIN {X 0,Y 228.461,Z 443.764,A -85,B 0,C 180,E1 -20092.649,E2 -20092.649} C_VEL
LIN {X 0,Y 230.051,Z 440.486,A -85,B 0,C 180,E1 -20095.322,E2 -20095.322} C_VEL
LIN {X 0,Y 232.018,Z 436.047,A -85,B 0,C 180,E1 -20098.003,E2 -20098.003} C_VEL
LIN {X 0,Y 234.493,Z 430.344,A -85,B 0,C 180,E1 -20100.632,E2 -20100.632} C_VEL
LIN {X 0,Y 237.374,Z 423.115,A -85,B 0,C 180,E1 -20103.212,E2 -20103.212} C_VEL
LIN {X 0,Y 240.618,Z 414.027,A -85,B 0,C 180,E1 -20105.744,E2 -20105.744} C_VEL
LIN {X 0,Y 243.672,Z 404.618,A -85,B 0,C 180,E1 -20107.799,E2 -20107.799} C_VEL
LIN {X 0,Y 246.676,Z 394.198,A -85,B 0,C 180,E1 -20109.573,E2 -20109.573} C_VEL
LIN {X 0,Y 249.437,Z 382.194,A -85,B 0,C 180,E1 -20111.192,E2 -20111.192} C_VEL
LIN {X 0,Y 251.559,Z 370.662,A -85,B 0,C 180,E1 -20112.375,E2 -20112.375} C_VEL
LIN {X 0,Y 253.486,Z 357.555,A -85,B 0,C 180,E1 -20113.329,E2 -20113.329} C_VEL
LIN {X 0,Y 254.72,Z 344.469,A -85,B 0,C 180,E1 -20113.972,E2 -20113.972} C_VEL
LIN {X 0,Y 257.315,Z 290.955,A -85,B 0,C 180,E1 -20115.444,E2 -20115.444} C_VEL
LIN {X 0,Y 250.714,Z 277.126,A -85,B 0,C 180,E1 -20117.202,E2 -20117.202} C_VEL
LIN {X 0,Y 246.438,Z 269.395,A -85,B 0,C 180,E1 -20118.373,E2 -20118.373} C_VEL
LIN {X 0,Y 238.945,Z 257.776,A -85,B 0,C 180,E1 -20120.51,E2 -20120.51} C_VEL
LIN {X 0,Y 236.213,Z 253.862,A -85,B 0,C 180,E1 -20121.331,E2 -20121.331} C_VEL
LIN {X 0,Y 233.687,Z 250.183,A -85,B 0,C 180,E1 -20122.121,E2 -20122.121} C_VEL
LIN {X 0,Y 231.383,Z 246.798,A -85,B 0,C 180,E1 -20122.869,E2 -20122.869} C_VEL
LIN {X 0,Y 230.689,Z 245.894,A -85,B 0,C 180,E1 -20123.094,E2 -20123.094} C_VEL
LIN {X 0,Y 228.716,Z 243.616,A -85,B 0,C 180,E1 -20123.733,E2 -20123.733} C_VEL
LIN {X 0,Y 227.903,Z 241.098,A -85,B 0,C 180,E1 -20124.132,E2 -20124.132} C_VEL
LIN {X 0,Y 227.865,Z 241.094,A -85,B 0,C 180,E1 -20128.377,E2 -20128.377} C_VEL
LIN {X 0,Y 227.879,Z 241.09,A -85,B 0,C 180,E1 -20132.444,E2 -20132.444} C_VEL
LIN {X 0,Y 227.898,Z 241.086,A -85,B 0,C 180,E1 -20136.365,E2 -20136.365} C_VEL
LIN {X 0,Y 227.915,Z 241.083,A -85,B 0,C 180,E1 -20140.172,E2 -20140.172} C_VEL
LIN {X 0,Y 228.02,Z 241.072,A -85,B 0,C 180,E1 -20143.895,E2 -20143.895} C_VEL
LIN {X 0,Y 228.117,Z 241.058,A -85,B 0,C 180,E1 -20149.347,E2 -20149.347} C_VEL
LIN {X 0,Y 228.306,Z 241.037,A -85,B 0,C 180,E1 -20152.927,E2 -20152.927} C_VEL
LIN {X 0,Y 228.537,Z 241.004,A -85,B 0,C 180,E1 -20158.238,E2 -20158.238} C_VEL
LIN {X 0,Y 228.529,Z 241.013,A -85,B 0,C 180,E1 -20161.762,E2 -20161.762} C_VEL
LIN {X 0,Y 228.281,Z 241.037,A -85,B 0,C 180,E1 -20167.074,E2 -20167.074} C_VEL
LIN {X 0,Y 228.117,Z 241.067,A -85,B 0,C 180,E1 -20170.652,E2 -20170.652} C_VEL
LIN {X 0,Y 228.019,Z 241.08,A -85,B 0,C 180,E1 -20174.275,E2 -20174.275} C_VEL
LIN {X 0,Y 227.896,Z 241.088,A -85,B 0,C 180,E1 -20178.268,E2 -20178.268} C_VEL
LIN {X 0,Y 227.881,Z 241.09,A -85,B 0,C 180,E1 -20182.304,E2 -20182.304} C_VEL
LIN {X 0,Y 227.854,Z 241.091,A -85,B 0,C 180,E1 -20185.939,E2 -20185.939} C_VEL
LIN {X 0,Y 227.175,Z 241.187,A -85,B 0,C 180,E1 -20187.415,E2 -20187.415} C_VEL
LIN {X 0,Y 224.298,Z 241.536,A -85,B 0,C 180,E1 -20189.822,E2 -20189.822} C_VEL
LIN {X 0,Y 221.871,Z 241.848,A -85,B 0,C 180,E1 -20191.787,E2 -20191.787} C_VEL
LIN {X 0,Y 220.853,Z 241.965,A -85,B 0,C 180,E1 -20193.313,E2 -20193.313} C_VEL
LIN {X 0,Y 220.783,Z 241.973,A -85,B 0,C 180,E1 -20193.83,E2 -20193.83} C_VEL
LIN {X 0,Y 220.785,Z 241.948,A -85,B 0,C 180,E1 -20198.368,E2 -20198.368} C_VEL
LIN {X 0,Y 220.772,Z 241.953,A -85,B 0,C 180,E1 -20199.249,E2 -20199.249} C_VEL
LIN {X 0,Y 223.027,Z 249.346,A -85,B 0,C 180,E1 -20203.889,E2 -20203.889} C_VEL
LIN {X 0,Y 224.057,Z 252.68,A -85,B 0,C 180,E1 -20205.791,E2 -20205.791} C_VEL
LIN {X 0,Y 226.717,Z 257.215,A -85,B 0,C 180,E1 -20206.759,E2 -20206.759} C_VEL
LIN {X 0,Y 228.554,Z 260.205,A -85,B 0,C 180,E1 -20207.398,E2 -20207.398} C_VEL
LIN {X 0,Y 231.796,Z 265.602,A -85,B 0,C 180,E1 -20208.488,E2 -20208.488} C_VEL
LIN {X 0,Y 236.665,Z 274.223,A -85,B 0,C 180,E1 -20210.055,E2 -20210.055} C_VEL
LIN {X 0,Y 243.157,Z 287.316,A -85,B 0,C 180,E1 -20212.047,E2 -20212.047} C_VEL
LIN {X 0,Y 248.074,Z 298.506,A -85,B 0,C 180,E1 -20213.492,E2 -20213.492} C_VEL
LIN {X 0,Y 250.667,Z 316.542,A -85,B 0,C 180,E1 -20214.666,E2 -20214.666} C_VEL
LIN {X 0,Y 248.349,Z 362.938,A -85,B 0,C 180,E1 -20215.972,E2 -20215.972} C_VEL
LIN {X 0,Y 246.864,Z 376.652,A -85,B 0,C 180,E1 -20216.64,E2 -20216.64} C_VEL
LIN {X 0,Y 244.653,Z 389.293,A -85,B 0,C 180,E1 -20217.532,E2 -20217.532} C_VEL
LIN {X 0,Y 241.969,Z 401.281,A -85,B 0,C 180,E1 -20218.722,E2 -20218.722} C_VEL
LIN {X 0,Y 238.914,Z 412.732,A -85,B 0,C 180,E1 -20220.237,E2 -20220.237} C_VEL
LIN {X 0,Y 235.624,Z 423.078,A -85,B 0,C 180,E1 -20221.979,E2 -20221.979} C_VEL
LIN {X 0,Y 232.408,Z 432.404,A -85,B 0,C 180,E1 -20223.992,E2 -20223.992} C_VEL
LIN {X 0,Y 228.878,Z 441.445,A -85,B 0,C 180,E1 -20226.472,E2 -20226.472} C_VEL
LIN {X 0,Y 226.067,Z 448.723,A -85,B 0,C 180,E1 -20229.037,E2 -20229.037} C_VEL
LIN {X 0,Y 223.625,Z 454.648,A -85,B 0,C 180,E1 -20231.681,E2 -20231.681} C_VEL
LIN {X 0,Y 221.657,Z 459.319,A -85,B 0,C 180,E1 -20234.363,E2 -20234.363} C_VEL
LIN {X 0,Y 220.168,Z 462.907,A -85,B 0,C 180,E1 -20237.086,E2 -20237.086} C_VEL
LIN {X 0,Y 219.53,Z 464.766,A -85,B 0,C 180,E1 -20238.923,E2 -20238.923} C_VEL
LIN {X 0,Y 218.694,Z 467.2,A -85,B 0,C 180,E1 -20242.612,E2 -20242.612} C_VEL
LIN {X 0,Y 218.596,Z 467.995,A -85,B 0,C 180,E1 -20245.323,E2 -20245.323} C_VEL
LIN {X 0,Y 218.734,Z 467.919,A -85,B 0,C 180,E1 -20248.155,E2 -20248.155} C_VEL
LIN {X 0,Y 218.811,Z 467.345,A -85,B 0,C 180,E1 -20249.997,E2 -20249.997} C_VEL
LIN {X 0,Y 218.768,Z 466.367,A -85,B 0,C 180,E1 -20251.837,E2 -20251.837} C_VEL
LIN {X 0,Y 218.647,Z 463.851,A -85,B 0,C 180,E1 -20254.836,E2 -20254.836} C_VEL
LIN {X 0,Y 218.826,Z 460.782,A -85,B 0,C 180,E1 -20257.377,E2 -20257.377} C_VEL
LIN {X 0,Y 219.191,Z 456.385,A -85,B 0,C 180,E1 -20260.153,E2 -20260.153} C_VEL
LIN {X 0,Y 219.872,Z 450.763,A -85,B 0,C 180,E1 -20262.924,E2 -20262.924} C_VEL
LIN {X 0,Y 221.217,Z 443.755,A -85,B 0,C 180,E1 -20265.662,E2 -20265.662} C_VEL
LIN {X 0,Y 222.806,Z 434.926,A -85,B 0,C 180,E1 -20268.381,E2 -20268.381} C_VEL
LIN {X 0,Y 224.568,Z 425.881,A -85,B 0,C 180,E1 -20270.609,E2 -20270.609} C_VEL
LIN {X 0,Y 226.394,Z 415.923,A -85,B 0,C 180,E1 -20272.586,E2 -20272.586} C_VEL
LIN {X 0,Y 228.316,Z 404.907,A -85,B 0,C 180,E1 -20274.306,E2 -20274.306} C_VEL
LIN {X 0,Y 230.191,Z 392.534,A -85,B 0,C 180,E1 -20275.783,E2 -20275.783} C_VEL
LIN {X 0,Y 231.615,Z 380.828,A -85,B 0,C 180,E1 -20276.824,E2 -20276.824} C_VEL
LIN {X 0,Y 232.786,Z 368.424,A -85,B 0,C 180,E1 -20277.59,E2 -20277.59} C_VEL
LIN {X 0,Y 233.513,Z 352.526,A -85,B 0,C 180,E1 -20278.167,E2 -20278.167} C_VEL
LIN {X 0,Y 234.801,Z 309.758,A -85,B 0,C 180,E1 -20279.443,E2 -20279.443} C_VEL
LIN {X 0,Y 230.933,Z 275.332,A -85,B 0,C 180,E1 -20281.055,E2 -20281.055} C_VEL
LIN {X 0,Y 230.051,Z 271.301,A -85,B 0,C 180,E1 -20281.302,E2 -20281.302} C_VEL
LIN {X 0,Y 223.694,Z 254.718,A -85,B 0,C 180,E1 -20282.731,E2 -20282.731} C_VEL
LIN {X 0,Y 221.386,Z 244.24,A -85,B 0,C 180,E1 -20287.088,E2 -20287.088} C_VEL
LIN {X 0,Y 220.846,Z 241.978,A -85,B 0,C 180,E1 -20288.129,E2 -20288.129} C_VEL
LIN {X 0,Y 220.749,Z 241.987,A -85,B 0,C 180,E1 -20292.924,E2 -20292.924} C_VEL
LIN {X 0,Y 220.842,Z 241.976,A -85,B 0,C 180,E1 -20297.038,E2 -20297.038} C_VEL
LIN {X 0,Y 220.832,Z 241.977,A -85,B 0,C 180,E1 -20300.469,E2 -20300.469} C_VEL
LIN {X 0,Y 220.777,Z 241.985,A -85,B 0,C 180,E1 -20305.041,E2 -20305.041} C_VEL
LIN {X 0,Y 220.841,Z 241.976,A -85,B 0,C 180,E1 -20309.391,E2 -20309.391} C_VEL
LIN {X 0,Y 220.866,Z 241.972,A -85,B 0,C 180,E1 -20313.546,E2 -20313.546} C_VEL
LIN {X 0,Y 220.911,Z 241.966,A -85,B 0,C 180,E1 -20317.557,E2 -20317.557} C_VEL
LIN {X 0,Y 220.95,Z 241.96,A -85,B 0,C 180,E1 -20322.571,E2 -20322.571} C_VEL
LIN {X 0,Y 220.969,Z 241.955,A -85,B 0,C 180,E1 -20327.136,E2 -20327.136} C_VEL
LIN {X 0,Y 221.171,Z 241.935,A -85,B 0,C 180,E1 -20330.858,E2 -20330.858} C_VEL
LIN {X 0,Y 221.224,Z 241.922,A -85,B 0,C 180,E1 -20332.7,E2 -20332.7} C_VEL
LIN {X 0,Y 221.472,Z 241.891,A -85,B 0,C 180,E1 -20338.182,E2 -20338.182} C_VEL
LIN {X 0,Y 221.445,Z 241.87,A -85,B 0,C 180,E1 -20341.819,E2 -20341.819} C_VEL
LIN {X 0,Y 221.214,Z 241.928,A -85,B 0,C 180,E1 -20347.301,E2 -20347.301} C_VEL
LIN {X 0,Y 221.026,Z 241.944,A -85,B 0,C 180,E1 -20350.999,E2 -20350.999} C_VEL
LIN {X 0,Y 220.942,Z 241.948,A -85,B 0,C 180,E1 -20356.636,E2 -20356.636} C_VEL
LIN {X 0,Y 220.817,Z 241.98,A -85,B 0,C 180,E1 -20360.494,E2 -20360.494} C_VEL
LIN {X 0,Y 220.828,Z 241.974,A -85,B 0,C 180,E1 -20364.44,E2 -20364.44} C_VEL
LIN {X 0,Y 220.797,Z 241.978,A -85,B 0,C 180,E1 -20368.519,E2 -20368.519} C_VEL
LIN {X 0,Y 220.79,Z 241.981,A -85,B 0,C 180,E1 -20372.761,E2 -20372.761} C_VEL
LIN {X 0,Y 220.816,Z 241.977,A -85,B 0,C 180,E1 -20377.293,E2 -20377.293} C_VEL
LIN {X 0,Y 220.83,Z 241.976,A -85,B 0,C 180,E1 -20381.939,E2 -20381.939} C_VEL
LIN {X 0,Y 220.764,Z 241.968,A -85,B 0,C 180,E1 -20385.554,E2 -20385.554} C_VEL
LIN {X 0,Y 220.77,Z 241.981,A -85,B 0,C 180,E1 -20390.464,E2 -20390.464} C_VEL
LIN {X 0,Y 220.81,Z 241.966,A -85,B 0,C 180,E1 -20392.799,E2 -20392.799} C_VEL
LIN {X 0,Y 220.804,Z 241.978,A -85,B 0,C 180,E1 -20397.249,E2 -20397.249} C_VEL
LIN {X 0,Y 220.817,Z 241.98,A -85,B 0,C 180,E1 -20401.491,E2 -20401.491} C_VEL
LIN {X 0,Y 220.854,Z 241.97,A -85,B 0,C 180,E1 -20405.57,E2 -20405.57} C_VEL
LIN {X 0,Y 220.918,Z 242.102,A -85,B 0,C 180,E1 -20408.174,E2 -20408.174} C_VEL
LIN {X 0,Y 221.927,Z 244.869,A -85,B 0,C 180,E1 -20408.417,E2 -20408.417} C_VEL
LIN {X 0,Y 229.657,Z 260.418,A -85,B 0,C 180,E1 -20409.996,E2 -20409.996} C_VEL
LIN {X 0,Y 233.362,Z 268.91,A -85,B 0,C 180,E1 -20410.745,E2 -20410.745} C_VEL
LIN {X 0,Y 235.893,Z 276.374,A -85,B 0,C 180,E1 -20411.296,E2 -20411.296} C_VEL
LIN {X 0,Y 233.457,Z 344.436,A -85,B 0,C 180,E1 -20413.331,E2 -20413.331} C_VEL
LIN {X 0,Y 232.498,Z 356.836,A -85,B 0,C 180,E1 -20413.993,E2 -20413.993} C_VEL
LIN {X 0,Y 231.442,Z 368.494,A -85,B 0,C 180,E1 -20414.934,E2 -20414.934} C_VEL
LIN {X 0,Y 230.297,Z 379.207,A -85,B 0,C 180,E1 -20416.099,E2 -20416.099} C_VEL
LIN {X 0,Y 228.6,Z 390.029,A -85,B 0,C 180,E1 -20417.577,E2 -20417.577} C_VEL
LIN {X 0,Y 226.889,Z 399.969,A -85,B 0,C 180,E1 -20419.294,E2 -20419.294} C_VEL
LIN {X 0,Y 224.908,Z 410.009,A -85,B 0,C 180,E1 -20421.468,E2 -20421.468} C_VEL
LIN {X 0,Y 223.113,Z 419.678,A -85,B 0,C 180,E1 -20424.128,E2 -20424.128} C_VEL
LIN {X 0,Y 221.501,Z 427.433,A -85,B 0,C 180,E1 -20426.821,E2 -20426.821} C_VEL
LIN {X 0,Y 220.52,Z 432.716,A -85,B 0,C 180,E1 -20429.09,E2 -20429.09} C_VEL
LIN {X 0,Y 219.692,Z 437.848,A -85,B 0,C 180,E1 -20431.836,E2 -20431.836} C_VEL
LIN {X 0,Y 219.195,Z 441.84,A -85,B 0,C 180,E1 -20434.601,E2 -20434.601} C_VEL
LIN {X 0,Y 218.767,Z 444.813,A -85,B 0,C 180,E1 -20437.386,E2 -20437.386} C_VEL
LIN {X 0,Y 218.579,Z 446.239,A -85,B 0,C 180,E1 -20439.254,E2 -20439.254} C_VEL
LIN {X 0,Y 218.656,Z 447.887,A -85,B 0,C 180,E1 -20443.005,E2 -20443.005} C_VEL
LIN {X 0,Y 219.059,Z 448.049,A -85,B 0,C 180,E1 -20445.743,E2 -20445.743} C_VEL
LIN {X 0,Y 219.709,Z 447.285,A -85,B 0,C 180,E1 -20448.657,E2 -20448.657} C_VEL
LIN {X 0,Y 220.363,Z 446.276,A -85,B 0,C 180,E1 -20450.539,E2 -20450.539} C_VEL
LIN {X 0,Y 221.549,Z 444.172,A -85,B 0,C 180,E1 -20453.081,E2 -20453.081} C_VEL
LIN {X 0,Y 223.435,Z 440.526,A -85,B 0,C 180,E1 -20456.128,E2 -20456.128} C_VEL
LIN {X 0,Y 225.457,Z 436.242,A -85,B 0,C 180,E1 -20458.741,E2 -20458.741} C_VEL
LIN {X 0,Y 228.2,Z 430.172,A -85,B 0,C 180,E1 -20461.572,E2 -20461.572} C_VEL
LIN {X 0,Y 231.279,Z 422.804,A -85,B 0,C 180,E1 -20464.206,E2 -20464.206} C_VEL
LIN {X 0,Y 234.126,Z 415.192,A -85,B 0,C 180,E1 -20466.378,E2 -20466.378} C_VEL
LIN {X 0,Y 237.256,Z 406.036,A -85,B 0,C 180,E1 -20468.467,E2 -20468.467} C_VEL
LIN {X 0,Y 240.396,Z 395.845,A -85,B 0,C 180,E1 -20470.292,E2 -20470.292} C_VEL
LIN {X 0,Y 243.268,Z 384.275,A -85,B 0,C 180,E1 -20471.918,E2 -20471.918} C_VEL
LIN {X 0,Y 245.617,Z 372.234,A -85,B 0,C 180,E1 -20473.23,E2 -20473.23} C_VEL
LIN {X 0,Y 247.626,Z 359.689,A -85,B 0,C 180,E1 -20474.195,E2 -20474.195} C_VEL
LIN {X 0,Y 249.028,Z 346.025,A -85,B 0,C 180,E1 -20474.91,E2 -20474.91} C_VEL
LIN {X 0,Y 251.651,Z 293.049,A -85,B 0,C 180,E1 -20476.427,E2 -20476.427} C_VEL
LIN {X 0,Y 244.848,Z 278.808,A -85,B 0,C 180,E1 -20478.343,E2 -20478.343} C_VEL
LIN {X 0,Y 237.329,Z 266.373,A -85,B 0,C 180,E1 -20480.533,E2 -20480.533} C_VEL
LIN {X 0,Y 232.443,Z 259.125,A -85,B 0,C 180,E1 -20482.047,E2 -20482.047} C_VEL
LIN {X 0,Y 229.241,Z 254.58,A -85,B 0,C 180,E1 -20483.088,E2 -20483.088} C_VEL
LIN {X 0,Y 226.936,Z 251.294,A -85,B 0,C 180,E1 -20483.87,E2 -20483.87} C_VEL
LIN {X 0,Y 224.708,Z 248.256,A -85,B 0,C 180,E1 -20484.647,E2 -20484.647} C_VEL
LIN {X 0,Y 223.959,Z 247.031,A -85,B 0,C 180,E1 -20484.924,E2 -20484.924} C_VEL
LIN {X 0,Y 221.764,Z 244.75,A -85,B 0,C 180,E1 -20485.693,E2 -20485.693} C_VEL
LIN {X 0,Y 220.842,Z 241.969,A -85,B 0,C 180,E1 -20486.161,E2 -20486.161} C_VEL
LIN {X 0,Y 220.865,Z 241.965,A -85,B 0,C 180,E1 -20489.394,E2 -20489.394} C_VEL
LIN {X 0,Y 220.888,Z 241.964,A -85,B 0,C 180,E1 -20493.548,E2 -20493.548} C_VEL
LIN {X 0,Y 220.855,Z 241.968,A -85,B 0,C 180,E1 -20497.551,E2 -20497.551} C_VEL
LIN {X 0,Y 220.937,Z 241.964,A -85,B 0,C 180,E1 -20502.605,E2 -20502.605} C_VEL
LIN {X 0,Y 220.977,Z 241.96,A -85,B 0,C 180,E1 -20507.136,E2 -20507.136} C_VEL
LIN {X 0,Y 221.179,Z 241.933,A -85,B 0,C 180,E1 -20510.858,E2 -20510.858} C_VEL
LIN {X 0,Y 221.241,Z 241.918,A -85,B 0,C 180,E1 -20512.7,E2 -20512.7} C_VEL
LIN {X 0,Y 221.495,Z 241.881,A -85,B 0,C 180,E1 -20518.182,E2 -20518.182} C_VEL
LIN {X 0,Y 221.462,Z 241.892,A -85,B 0,C 180,E1 -20521.818,E2 -20521.818} C_VEL
LIN {X 0,Y 221.218,Z 241.915,A -85,B 0,C 180,E1 -20527.301,E2 -20527.301} C_VEL
LIN {X 0,Y 221.043,Z 241.945,A -85,B 0,C 180,E1 -20530.998,E2 -20530.998} C_VEL
LIN {X 0,Y 220.967,Z 241.948,A -85,B 0,C 180,E1 -20536.634,E2 -20536.634} C_VEL
LIN {X 0,Y 220.84,Z 241.967,A -85,B 0,C 180,E1 -20540.491,E2 -20540.491} C_VEL
LIN {X 0,Y 220.793,Z 241.977,A -85,B 0,C 180,E1 -20544.444,E2 -20544.444} C_VEL
LIN {X 0,Y 220.783,Z 241.979,A -85,B 0,C 180,E1 -20548.521,E2 -20548.521} C_VEL
LIN {X 0,Y 220.796,Z 241.974,A -85,B 0,C 180,E1 -20552.76,E2 -20552.76} C_VEL
LIN {X 0,Y 220.783,Z 241.973,A -85,B 0,C 180,E1 -20553.83,E2 -20553.83} C_VEL
LIN {X 0,Y 220.12,Z 242.083,A -85,B 0,C 180,E1 -20554.858,E2 -20554.858} C_VEL
LIN {X 0,Y 217.334,Z 242.754,A -85,B 0,C 180,E1 -20556.477,E2 -20556.477} C_VEL
LIN {X 0,Y 214.781,Z 244.156,A -85,B 0,C 180,E1 -20558.1,E2 -20558.1} C_VEL
LIN {X 0,Y 214.486,Z 245.416,A -85,B 0,C 180,E1 -20559.107,E2 -20559.107} C_VEL
LIN {X 0,Y 216.58,Z 252.025,A -85,B 0,C 180,E1 -20563.43,E2 -20563.43} C_VEL
LIN {X 0,Y 219.291,Z 256.573,A -85,B 0,C 180,E1 -20564.55,E2 -20564.55} C_VEL
LIN {X 0,Y 220.853,Z 258.894,A -85,B 0,C 180,E1 -20565.145,E2 -20565.145} C_VEL
LIN {X 0,Y 224.972,Z 265.686,A -85,B 0,C 180,E1 -20566.668,E2 -20566.668} C_VEL
LIN {X 0,Y 229.97,Z 274.164,A -85,B 0,C 180,E1 -20568.398,E2 -20568.398} C_VEL
LIN {X 0,Y 236.102,Z 286.09,A -85,B 0,C 180,E1 -20570.418,E2 -20570.418} C_VEL
LIN {X 0,Y 242.821,Z 301.171,A -85,B 0,C 180,E1 -20572.519,E2 -20572.519} C_VEL
LIN {X 0,Y 245.178,Z 317.628,A -85,B 0,C 180,E1 -20573.639,E2 -20573.639} C_VEL
LIN {X 0,Y 242.806,Z 362.862,A -85,B 0,C 180,E1 -20574.937,E2 -20574.937} C_VEL
LIN {X 0,Y 241.288,Z 376.361,A -85,B 0,C 180,E1 -20575.607,E2 -20575.607} C_VEL
LIN {X 0,Y 238.959,Z 389.259,A -85,B 0,C 180,E1 -20576.533,E2 -20576.533} C_VEL
LIN {X 0,Y 236.349,Z 400.375,A -85,B 0,C 180,E1 -20577.639,E2 -20577.639} C_VEL
LIN {X 0,Y 233.188,Z 411.929,A -85,B 0,C 180,E1 -20579.178,E2 -20579.178} C_VEL
LIN {X 0,Y 229.755,Z 422.356,A -85,B 0,C 180,E1 -20580.947,E2 -20580.947} C_VEL
LIN {X 0,Y 226.692,Z 430.893,A -85,B 0,C 180,E1 -20582.787,E2 -20582.787} C_VEL
LIN {X 0,Y 223.551,Z 438.79,A -85,B 0,C 180,E1 -20584.885,E2 -20584.885} C_VEL
LIN {X 0,Y 220.332,Z 446.542,A -85,B 0,C 180,E1 -20587.493,E2 -20587.493} C_VEL
LIN {X 0,Y 217.705,Z 452.784,A -85,B 0,C 180,E1 -20590.185,E2 -20590.185} C_VEL
LIN {X 0,Y 215.473,Z 457.777,A -85,B 0,C 180,E1 -20592.928,E2 -20592.928} C_VEL
LIN {X 0,Y 213.668,Z 461.663,A -85,B 0,C 180,E1 -20595.716,E2 -20595.716} C_VEL
LIN {X 0,Y 212.518,Z 464.552,A -85,B 0,C 180,E1 -20598.553,E2 -20598.553} C_VEL
LIN {X 0,Y 211.634,Z 466.934,A -85,B 0,C 180,E1 -20602.364,E2 -20602.364} C_VEL
LIN {X 0,Y 211.514,Z 467.707,A -85,B 0,C 180,E1 -20605.424,E2 -20605.424} C_VEL
LIN {X 0,Y 211.641,Z 467.554,A -85,B 0,C 180,E1 -20608.094,E2 -20608.094} C_VEL
LIN {X 0,Y 211.743,Z 466.957,A -85,B 0,C 180,E1 -20609.996,E2 -20609.996} C_VEL
LIN {X 0,Y 211.675,Z 465.953,A -85,B 0,C 180,E1 -20611.899,E2 -20611.899} C_VEL
LIN {X 0,Y 211.554,Z 463.661,A -85,B 0,C 180,E1 -20614.706,E2 -20614.706} C_VEL
LIN {X 0,Y 211.741,Z 460.26,A -85,B 0,C 180,E1 -20617.625,E2 -20617.625} C_VEL
LIN {X 0,Y 212.143,Z 455.802,A -85,B 0,C 180,E1 -20620.494,E2 -20620.494} C_VEL
LIN {X 0,Y 212.925,Z 450.119,A -85,B 0,C 180,E1 -20623.354,E2 -20623.354} C_VEL
LIN {X 0,Y 214.323,Z 443.01,A -85,B 0,C 180,E1 -20626.179,E2 -20626.179} C_VEL
LIN {X 0,Y 215.747,Z 435.738,A -85,B 0,C 180,E1 -20628.513,E2 -20628.513} C_VEL
LIN {X 0,Y 217.22,Z 428.128,A -85,B 0,C 180,E1 -20630.535,E2 -20630.535} C_VEL
LIN {X 0,Y 219.113,Z 418.409,A -85,B 0,C 180,E1 -20632.631,E2 -20632.631} C_VEL
LIN {X 0,Y 221.029,Z 408.082,A -85,B 0,C 180,E1 -20634.41,E2 -20634.41} C_VEL
LIN {X 0,Y 222.947,Z 396.795,A -85,B 0,C 180,E1 -20635.931,E2 -20635.931} C_VEL
LIN {X 0,Y 224.575,Z 385.354,A -85,B 0,C 180,E1 -20637.105,E2 -20637.105} C_VEL
LIN {X 0,Y 225.815,Z 373.339,A -85,B 0,C 180,E1 -20638.003,E2 -20638.003} C_VEL
LIN {X 0,Y 226.795,Z 359.447,A -85,B 0,C 180,E1 -20638.653,E2 -20638.653} C_VEL
LIN {X 0,Y 228.403,Z 311.02,A -85,B 0,C 180,E1 -20640.137,E2 -20640.137} C_VEL
LIN {X 0,Y 224.669,Z 276.962,A -85,B 0,C 180,E1 -20641.788,E2 -20641.788} C_VEL
LIN {X 0,Y 224.048,Z 274.027,A -85,B 0,C 180,E1 -20641.973,E2 -20641.973} C_VEL
LIN {X 0,Y 217.527,Z 257.321,A -85,B 0,C 180,E1 -20643.471,E2 -20643.471} C_VEL
LIN {X 0,Y 216.405,Z 254.246,A -85,B 0,C 180,E1 -20643.807,E2 -20643.807} C_VEL
LIN {X 0,Y 214.222,Z 244.479,A -85,B 0,C 180,E1 -20648.059,E2 -20648.059} C_VEL
LIN {X 0,Y 213.761,Z 242.86,A -85,B 0,C 180,E1 -20648.876,E2 -20648.876} C_VEL
LIN {X 0,Y 213.692,Z 242.868,A -85,B 0,C 180,E1 -20653.672,E2 -20653.672} C_VEL
LIN {X 0,Y 213.759,Z 242.859,A -85,B 0,C 180,E1 -20656.335,E2 -20656.335} C_VEL
LIN {X 0,Y 213.772,Z 242.858,A -85,B 0,C 180,E1 -20659.114,E2 -20659.114} C_VEL
LIN {X 0,Y 213.72,Z 242.864,A -85,B 0,C 180,E1 -20663.707,E2 -20663.707} C_VEL
LIN {X 0,Y 213.754,Z 242.859,A -85,B 0,C 180,E1 -20668.727,E2 -20668.727} C_VEL
LIN {X 0,Y 213.798,Z 242.852,A -85,B 0,C 180,E1 -20672.599,E2 -20672.599} C_VEL
LIN {X 0,Y 213.839,Z 242.847,A -85,B 0,C 180,E1 -20676.939,E2 -20676.939} C_VEL
LIN {X 0,Y 213.899,Z 242.838,A -85,B 0,C 180,E1 -20682.305,E2 -20682.305} C_VEL
LIN {X 0,Y 213.91,Z 242.833,A -85,B 0,C 180,E1 -20686.704,E2 -20686.704} C_VEL
LIN {X 0,Y 214.108,Z 242.814,A -85,B 0,C 180,E1 -20690.554,E2 -20690.554} C_VEL
LIN {X 0,Y 214.063,Z 242.816,A -85,B 0,C 180,E1 -20694.348,E2 -20694.348} C_VEL
LIN {X 0,Y 214.406,Z 242.772,A -85,B 0,C 180,E1 -20698.122,E2 -20698.122} C_VEL
LIN {X 0,Y 214.505,Z 242.749,A -85,B 0,C 180,E1 -20700,E2 -20700} C_VEL
LIN {X 0,Y 214.382,Z 242.749,A -85,B 0,C 180,E1 -20701.879,E2 -20701.879} C_VEL
LIN {X 0,Y 214.153,Z 242.807,A -85,B 0,C 180,E1 -20707.543,E2 -20707.543} C_VEL
LIN {X 0,Y 213.956,Z 242.822,A -85,B 0,C 180,E1 -20711.367,E2 -20711.367} C_VEL
LIN {X 0,Y 213.847,Z 242.822,A -85,B 0,C 180,E1 -20715.243,E2 -20715.243} C_VEL
LIN {X 0,Y 213.762,Z 242.857,A -85,B 0,C 180,E1 -20719.195,E2 -20719.195} C_VEL
LIN {X 0,Y 213.766,Z 242.851,A -85,B 0,C 180,E1 -20723.237,E2 -20723.237} C_VEL
LIN {X 0,Y 213.802,Z 242.85,A -85,B 0,C 180,E1 -20727.454,E2 -20727.454} C_VEL
LIN {X 0,Y 213.741,Z 242.86,A -85,B 0,C 180,E1 -20731.742,E2 -20731.742} C_VEL
LIN {X 0,Y 213.721,Z 242.863,A -85,B 0,C 180,E1 -20736.293,E2 -20736.293} C_VEL
LIN {X 0,Y 213.773,Z 242.854,A -85,B 0,C 180,E1 -20740.886,E2 -20740.886} C_VEL
LIN {X 0,Y 213.76,Z 242.851,A -85,B 0,C 180,E1 -20743.682,E2 -20743.682} C_VEL
LIN {X 0,Y 213.69,Z 242.864,A -85,B 0,C 180,E1 -20748.879,E2 -20748.879} C_VEL
LIN {X 0,Y 213.73,Z 242.85,A -85,B 0,C 180,E1 -20753.717,E2 -20753.717} C_VEL
LIN {X 0,Y 213.77,Z 242.856,A -85,B 0,C 180,E1 -20758.737,E2 -20758.737} C_VEL
LIN {X 0,Y 213.818,Z 242.85,A -85,B 0,C 180,E1 -20762.609,E2 -20762.609} C_VEL
LIN {X 0,Y 213.82,Z 242.846,A -85,B 0,C 180,E1 -20767.125,E2 -20767.125} C_VEL
LIN {X 0,Y 214.974,Z 245.906,A -85,B 0,C 180,E1 -20767.45,E2 -20767.45} C_VEL
LIN {X 0,Y 222.215,Z 260.132,A -85,B 0,C 180,E1 -20769.007,E2 -20769.007} C_VEL
LIN {X 0,Y 227.398,Z 271.703,A -85,B 0,C 180,E1 -20770.102,E2 -20770.102} C_VEL
LIN {X 0,Y 229.531,Z 278.036,A -85,B 0,C 180,E1 -20770.589,E2 -20770.589} C_VEL
LIN {X 0,Y 226.996,Z 344.412,A -85,B 0,C 180,E1 -20772.61,E2 -20772.61} C_VEL
LIN {X 0,Y 225.978,Z 356.94,A -85,B 0,C 180,E1 -20773.286,E2 -20773.286} C_VEL
LIN {X 0,Y 224.899,Z 368.647,A -85,B 0,C 180,E1 -20774.253,E2 -20774.253} C_VEL
LIN {X 0,Y 223.466,Z 381.15,A -85,B 0,C 180,E1 -20775.665,E2 -20775.665} C_VEL
LIN {X 0,Y 221.45,Z 392.919,A -85,B 0,C 180,E1 -20777.402,E2 -20777.402} C_VEL
LIN {X 0,Y 219.53,Z 403.431,A -85,B 0,C 180,E1 -20779.397,E2 -20779.397} C_VEL
LIN {X 0,Y 217.572,Z 412.926,A -85,B 0,C 180,E1 -20781.646,E2 -20781.646} C_VEL
LIN {X 0,Y 215.794,Z 422.029,A -85,B 0,C 180,E1 -20784.397,E2 -20784.397} C_VEL
LIN {X 0,Y 214.207,Z 429.388,A -85,B 0,C 180,E1 -20787.183,E2 -20787.183} C_VEL
LIN {X 0,Y 213.144,Z 435.278,A -85,B 0,C 180,E1 -20790.004,E2 -20790.004} C_VEL
LIN {X 0,Y 212.355,Z 439.938,A -85,B 0,C 180,E1 -20792.849,E2 -20792.849} C_VEL
LIN {X 0,Y 211.946,Z 443.65,A -85,B 0,C 180,E1 -20795.852,E2 -20795.852} C_VEL
LIN {X 0,Y 211.634,Z 445.322,A -85,B 0,C 180,E1 -20797.636,E2 -20797.636} C_VEL
LIN {X 0,Y 211.47,Z 446.701,A -85,B 0,C 180,E1 -20799.568,E2 -20799.568} C_VEL
LIN {X 0,Y 211.627,Z 448.273,A -85,B 0,C 180,E1 -20803.445,E2 -20803.445} C_VEL
LIN {X 0,Y 212.001,Z 448.384,A -85,B 0,C 180,E1 -20805.975,E2 -20805.975} C_VEL
LIN {X 0,Y 212.803,Z 447.525,A -85,B 0,C 180,E1 -20809.286,E2 -20809.286} C_VEL
LIN {X 0,Y 213.549,Z 446.465,A -85,B 0,C 180,E1 -20811.226,E2 -20811.226} C_VEL
LIN {X 0,Y 214.664,Z 444.572,A -85,B 0,C 180,E1 -20813.55,E2 -20813.55} C_VEL
LIN {X 0,Y 216.864,Z 440.56,A -85,B 0,C 180,E1 -20816.983,E2 -20816.983} C_VEL
LIN {X 0,Y 219.512,Z 435.186,A -85,B 0,C 180,E1 -20820.18,E2 -20820.18} C_VEL
LIN {X 0,Y 222.513,Z 428.84,A -85,B 0,C 180,E1 -20823.014,E2 -20823.014} C_VEL
LIN {X 0,Y 225.832,Z 421.103,A -85,B 0,C 180,E1 -20825.698,E2 -20825.698} C_VEL
LIN {X 0,Y 228.88,Z 413.095,A -85,B 0,C 180,E1 -20827.888,E2 -20827.888} C_VEL
LIN {X 0,Y 232.282,Z 403.252,A -85,B 0,C 180,E1 -20830.012,E2 -20830.012} C_VEL
LIN {X 0,Y 235.695,Z 392.038,A -85,B 0,C 180,E1 -20831.895,E2 -20831.895} C_VEL
LIN {X 0,Y 238.21,Z 381.397,A -85,B 0,C 180,E1 -20833.31,E2 -20833.31} C_VEL
LIN {X 0,Y 240.354,Z 370.53,A -85,B 0,C 180,E1 -20834.421,E2 -20834.421} C_VEL
LIN {X 0,Y 242.424,Z 357.149,A -85,B 0,C 180,E1 -20835.403,E2 -20835.403} C_VEL
LIN {X 0,Y 243.637,Z 344.83,A -85,B 0,C 180,E1 -20836.011,E2 -20836.011} C_VEL
LIN {X 0,Y 246.273,Z 295.553,A -85,B 0,C 180,E1 -20837.399,E2 -20837.399} C_VEL
LIN {X 0,Y 239.49,Z 281.5,A -85,B 0,C 180,E1 -20839.408,E2 -20839.408} C_VEL
LIN {X 0,Y 231.43,Z 268.357,A -85,B 0,C 180,E1 -20841.9,E2 -20841.9} C_VEL
LIN {X 0,Y 225.853,Z 260.251,A -85,B 0,C 180,E1 -20843.755,E2 -20843.755} C_VEL
LIN {X 0,Y 223.283,Z 256.641,A -85,B 0,C 180,E1 -20844.659,E2 -20844.659} C_VEL
LIN {X 0,Y 220.459,Z 252.676,A -85,B 0,C 180,E1 -20845.7,E2 -20845.7} C_VEL
LIN {X 0,Y 218.038,Z 249.653,A -85,B 0,C 180,E1 -20846.615,E2 -20846.615} C_VEL
LIN {X 0,Y 217.324,Z 248.124,A -85,B 0,C 180,E1 -20846.926,E2 -20846.926} C_VEL
LIN {X 0,Y 215.057,Z 246.16,A -85,B 0,C 180,E1 -20847.785,E2 -20847.785} C_VEL
LIN {X 0,Y 213.892,Z 243.641,A -85,B 0,C 180,E1 -20848.323,E2 -20848.323} C_VEL
LIN {X 0,Y 213.749,Z 242.852,A -85,B 0,C 180,E1 -20848.42,E2 -20848.42} C_VEL
LIN {X 0,Y 213.823,Z 242.84,A -85,B 0,C 180,E1 -20852.602,E2 -20852.602} C_VEL
LIN {X 0,Y 213.812,Z 242.841,A -85,B 0,C 180,E1 -20856.974,E2 -20856.974} C_VEL
LIN {X 0,Y 213.9,Z 242.841,A -85,B 0,C 180,E1 -20862.8,E2 -20862.8} C_VEL
LIN {X 0,Y 213.916,Z 242.839,A -85,B 0,C 180,E1 -20866.704,E2 -20866.704} C_VEL
LIN {X 0,Y 214.118,Z 242.81,A -85,B 0,C 180,E1 -20870.554,E2 -20870.554} C_VEL
LIN {X 0,Y 214.08,Z 242.808,A -85,B 0,C 180,E1 -20874.348,E2 -20874.348} C_VEL
LIN {X 0,Y 214.428,Z 242.761,A -85,B 0,C 180,E1 -20878.122,E2 -20878.122} C_VEL
LIN {X 0,Y 214.527,Z 242.759,A -85,B 0,C 180,E1 -20880,E2 -20880} C_VEL
LIN {X 0,Y 214.399,Z 242.77,A -85,B 0,C 180,E1 -20881.878,E2 -20881.878} C_VEL
LIN {X 0,Y 214.16,Z 242.794,A -85,B 0,C 180,E1 -20887.543,E2 -20887.543} C_VEL
LIN {X 0,Y 213.977,Z 242.821,A -85,B 0,C 180,E1 -20891.365,E2 -20891.365} C_VEL
LIN {X 0,Y 213.886,Z 242.84,A -85,B 0,C 180,E1 -20895.24,E2 -20895.24} C_VEL
LIN {X 0,Y 213.785,Z 242.855,A -85,B 0,C 180,E1 -20899.192,E2 -20899.192} C_VEL
LIN {X 0,Y 213.778,Z 242.855,A -85,B 0,C 180,E1 -20903.235,E2 -20903.235} C_VEL
LIN {X 0,Y 213.762,Z 242.857,A -85,B 0,C 180,E1 -20907.418,E2 -20907.418} C_VEL
LIN {X 0,Y 213.75,Z 242.86,A -85,B 0,C 180,E1 -20911.74,E2 -20911.74} C_VEL
LIN {X 0,Y 213.736,Z 242.846,A -85,B 0,C 180,E1 -20916.29,E2 -20916.29} C_VEL
LIN {X 0,Y 213.776,Z 243.036,A -85,B 0,C 180,E1 -20917.433,E2 -20917.433} C_VEL
LIN {X 0,Y 214.486,Z 245.416,A -85,B 0,C 180,E1 -20919.107,E2 -20919.107} C_VEL
LIN {X 0,Y 214.85,Z 247.2,A -85,B 0,C 180,E1 -20920.034,E2 -20920.034} C_VEL
LIN {X 0,Y 215.131,Z 250.945,A -85,B 0,C 180,E1 -20921.255,E2 -20921.255} C_VEL
LIN {X 0,Y 215.4,Z 255.388,A -85,B 0,C 180,E1 -20922.319,E2 -20922.319} C_VEL
LIN {X 0,Y 216.856,Z 263.111,A -85,B 0,C 180,E1 -20923.972,E2 -20923.972} C_VEL
LIN {X 0,Y 219.022,Z 267.073,A -85,B 0,C 180,E1 -20924.993,E2 -20924.993} C_VEL
LIN {X 0,Y 224.141,Z 275.823,A -85,B 0,C 180,E1 -20926.911,E2 -20926.911} C_VEL
LIN {X 0,Y 230.023,Z 286.812,A -85,B 0,C 180,E1 -20928.97,E2 -20928.97} C_VEL
LIN {X 0,Y 236.58,Z 301.37,A -85,B 0,C 180,E1 -20931.162,E2 -20931.162} C_VEL
LIN {X 0,Y 237.976,Z 305.145,A -85,B 0,C 180,E1 -20931.629,E2 -20931.629} C_VEL
LIN {X 0,Y 239.794,Z 318.786,A -85,B 0,C 180,E1 -20932.57,E2 -20932.57} C_VEL
LIN {X 0,Y 237.403,Z 362.219,A -85,B 0,C 180,E1 -20933.827,E2 -20933.827} C_VEL
LIN {X 0,Y 235.889,Z 375.426,A -85,B 0,C 180,E1 -20934.481,E2 -20934.481} C_VEL
LIN {X 0,Y 233.566,Z 388.149,A -85,B 0,C 180,E1 -20935.393,E2 -20935.393} C_VEL
LIN {X 0,Y 230.886,Z 399.477,A -85,B 0,C 180,E1 -20936.515,E2 -20936.515} C_VEL
LIN {X 0,Y 227.952,Z 409.861,A -85,B 0,C 180,E1 -20937.87,E2 -20937.87} C_VEL
LIN {X 0,Y 224.317,Z 420.584,A -85,B 0,C 180,E1 -20939.654,E2 -20939.654} C_VEL
LIN {X 0,Y 220.417,Z 431.132,A -85,B 0,C 180,E1 -20941.945,E2 -20941.945} C_VEL
LIN {X 0,Y 216.524,Z 440.289,A -85,B 0,C 180,E1 -20944.527,E2 -20944.527} C_VEL
LIN {X 0,Y 213.772,Z 446.565,A -85,B 0,C 180,E1 -20946.763,E2 -20946.763} C_VEL
LIN {X 0,Y 211.032,Z 452.74,A -85,B 0,C 180,E1 -20949.53,E2 -20949.53} C_VEL
LIN {X 0,Y 208.671,Z 457.672,A -85,B 0,C 180,E1 -20952.353,E2 -20952.353} C_VEL
LIN {X 0,Y 206.755,Z 461.501,A -85,B 0,C 180,E1 -20955.228,E2 -20955.228} C_VEL
LIN {X 0,Y 205.523,Z 464.336,A -85,B 0,C 180,E1 -20958.158,E2 -20958.158} C_VEL
LIN {X 0,Y 204.595,Z 466.669,A -85,B 0,C 180,E1 -20962.099,E2 -20962.099} C_VEL
LIN {X 0,Y 204.44,Z 467.418,A -85,B 0,C 180,E1 -20965.51,E2 -20965.51} C_VEL
LIN {X 0,Y 204.55,Z 467.189,A -85,B 0,C 180,E1 -20968.028,E2 -20968.028} C_VEL
LIN {X 0,Y 204.675,Z 466.568,A -85,B 0,C 180,E1 -20969.996,E2 -20969.996} C_VEL
LIN {X 0,Y 204.585,Z 465.536,A -85,B 0,C 180,E1 -20971.965,E2 -20971.965} C_VEL
LIN {X 0,Y 204.465,Z 463.456,A -85,B 0,C 180,E1 -20974.58,E2 -20974.58} C_VEL
LIN {X 0,Y 204.673,Z 459.734,A -85,B 0,C 180,E1 -20977.89,E2 -20977.89} C_VEL
LIN {X 0,Y 205.112,Z 455.216,A -85,B 0,C 180,E1 -20980.858,E2 -20980.858} C_VEL
LIN {X 0,Y 206.214,Z 448.352,A -85,B 0,C 180,E1 -20984.3,E2 -20984.3} C_VEL
LIN {X 0,Y 207.678,Z 440.868,A -85,B 0,C 180,E1 -20987.218,E2 -20987.218} C_VEL
LIN {X 0,Y 208.875,Z 434.877,A -85,B 0,C 180,E1 -20989.145,E2 -20989.145} C_VEL
LIN {X 0,Y 210.816,Z 425.959,A -85,B 0,C 180,E1 -20991.507,E2 -20991.507} C_VEL
LIN {X 0,Y 212.774,Z 416.145,A -85,B 0,C 180,E1 -20993.603,E2 -20993.603} C_VEL
LIN {X 0,Y 214.525,Z 406.842,A -85,B 0,C 180,E1 -20995.2,E2 -20995.2} C_VEL
LIN {X 0,Y 216.547,Z 395.338,A -85,B 0,C 180,E1 -20996.757,E2 -20996.757} C_VEL
LIN {X 0,Y 218.237,Z 383.432,A -85,B 0,C 180,E1 -20997.96,E2 -20997.96} C_VEL
LIN {X 0,Y 219.604,Z 370.186,A -85,B 0,C 180,E1 -20998.905,E2 -20998.905} C_VEL
LIN {X 0,Y 220.372,Z 357.689,A -85,B 0,C 180,E1 -20999.465,E2 -20999.465} C_VEL
LIN {X 0,Y 221.901,Z 310.764,A -85,B 0,C 180,E1 -21000.943,E2 -21000.943} C_VEL
LIN {X 0,Y 218.307,Z 277.675,A -85,B 0,C 180,E1 -21002.614,E2 -21002.614} C_VEL
LIN {X 0,Y 213.674,Z 265.022,A -85,B 0,C 180,E1 -21003.744,E2 -21003.744} C_VEL
LIN {X 0,Y 209.115,Z 253.96,A -85,B 0,C 180,E1 -21004.89,E2 -21004.89} C_VEL
LIN {X 0,Y 207.165,Z 245.581,A -85,B 0,C 180,E1 -21008.715,E2 -21008.715} C_VEL
LIN {X 0,Y 206.734,Z 243.735,A -85,B 0,C 180,E1 -21009.664,E2 -21009.664} C_VEL
LIN {X 0,Y 206.661,Z 243.742,A -85,B 0,C 180,E1 -21015.563,E2 -21015.563} C_VEL
LIN {X 0,Y 206.702,Z 243.738,A -85,B 0,C 180,E1 -21019.758,E2 -21019.758} C_VEL
LIN {X 0,Y 206.7,Z 243.738,A -85,B 0,C 180,E1 -21022.265,E2 -21022.265} C_VEL
LIN {X 0,Y 206.673,Z 243.74,A -85,B 0,C 180,E1 -21027.038,E2 -21027.038} C_VEL
LIN {X 0,Y 206.739,Z 243.732,A -85,B 0,C 180,E1 -21032.093,E2 -21032.093} C_VEL
LIN {X 0,Y 206.769,Z 243.727,A -85,B 0,C 180,E1 -21036.573,E2 -21036.573} C_VEL
LIN {X 0,Y 206.856,Z 243.716,A -85,B 0,C 180,E1 -21042.017,E2 -21042.017} C_VEL
LIN {X 0,Y 206.853,Z 243.712,A -85,B 0,C 180,E1 -21046.242,E2 -21046.242} C_VEL
LIN {X 0,Y 207.067,Z 243.69,A -85,B 0,C 180,E1 -21050.23,E2 -21050.23} C_VEL
LIN {X 0,Y 207.025,Z 243.693,A -85,B 0,C 180,E1 -21054.155,E2 -21054.155} C_VEL
LIN {X 0,Y 207.343,Z 243.651,A -85,B 0,C 180,E1 -21058.058,E2 -21058.058} C_VEL
LIN {X 0,Y 207.471,Z 243.624,A -85,B 0,C 180,E1 -21060,E2 -21060} C_VEL
LIN {X 0,Y 207.033,Z 243.676,A -85,B 0,C 180,E1 -21063.893,E2 -21063.893} C_VEL
LIN {X 0,Y 207.095,Z 243.686,A -85,B 0,C 180,E1 -21067.802,E2 -21067.802} C_VEL
LIN {X 0,Y 206.877,Z 243.703,A -85,B 0,C 180,E1 -21071.761,E2 -21071.761} C_VEL
LIN {X 0,Y 206.779,Z 243.705,A -85,B 0,C 180,E1 -21075.778,E2 -21075.778} C_VEL
LIN {X 0,Y 206.682,Z 243.738,A -85,B 0,C 180,E1 -21079.88,E2 -21079.88} C_VEL
LIN {X 0,Y 206.71,Z 243.73,A -85,B 0,C 180,E1 -21084.079,E2 -21084.079} C_VEL
LIN {X 0,Y 206.71,Z 243.732,A -85,B 0,C 180,E1 -21088.424,E2 -21088.424} C_VEL
LIN {X 0,Y 206.674,Z 243.738,A -85,B 0,C 180,E1 -21092.963,E2 -21092.963} C_VEL
LIN {X 0,Y 206.701,Z 243.736,A -85,B 0,C 180,E1 -21097.736,E2 -21097.736} C_VEL
LIN {X 0,Y 206.697,Z 243.735,A -85,B 0,C 180,E1 -21101.592,E2 -21101.592} C_VEL
LIN {X 0,Y 206.62,Z 243.728,A -85,B 0,C 180,E1 -21105.586,E2 -21105.586} C_VEL
LIN {X 0,Y 206.637,Z 243.743,A -85,B 0,C 180,E1 -21109.753,E2 -21109.753} C_VEL
LIN {X 0,Y 206.686,Z 243.735,A -85,B 0,C 180,E1 -21114.695,E2 -21114.695} C_VEL
LIN {X 0,Y 206.696,Z 243.738,A -85,B 0,C 180,E1 -21119.342,E2 -21119.342} C_VEL
LIN {X 0,Y 206.723,Z 243.735,A -85,B 0,C 180,E1 -21123.778,E2 -21123.778} C_VEL
LIN {X 0,Y 206.739,Z 243.731,A -85,B 0,C 180,E1 -21126.073,E2 -21126.073} C_VEL
LIN {X 0,Y 207.723,Z 246.556,A -85,B 0,C 180,E1 -21126.346,E2 -21126.346} C_VEL
LIN {X 0,Y 209.61,Z 249.858,A -85,B 0,C 180,E1 -21126.777,E2 -21126.777} C_VEL
LIN {X 0,Y 216.797,Z 264.099,A -85,B 0,C 180,E1 -21128.398,E2 -21128.398} C_VEL
LIN {X 0,Y 221.53,Z 274.865,A -85,B 0,C 180,E1 -21129.446,E2 -21129.446} C_VEL
LIN {X 0,Y 223.1,Z 279.932,A -85,B 0,C 180,E1 -21129.836,E2 -21129.836} C_VEL
LIN {X 0,Y 220.476,Z 345.541,A -85,B 0,C 180,E1 -21131.898,E2 -21131.898} C_VEL
LIN {X 0,Y 219.419,Z 358.527,A -85,B 0,C 180,E1 -21132.651,E2 -21132.651} C_VEL
LIN {X 0,Y 218.389,Z 368.799,A -85,B 0,C 180,E1 -21133.53,E2 -21133.53} C_VEL
LIN {X 0,Y 216.887,Z 381.343,A -85,B 0,C 180,E1 -21134.981,E2 -21134.981} C_VEL
LIN {X 0,Y 214.795,Z 393.145,A -85,B 0,C 180,E1 -21136.765,E2 -21136.765} C_VEL
LIN {X 0,Y 212.795,Z 403.674,A -85,B 0,C 180,E1 -21138.816,E2 -21138.816} C_VEL
LIN {X 0,Y 210.918,Z 412.301,A -85,B 0,C 180,E1 -21140.898,E2 -21140.898} C_VEL
LIN {X 0,Y 209.316,Z 420.218,A -85,B 0,C 180,E1 -21143.256,E2 -21143.256} C_VEL
LIN {X 0,Y 207.564,Z 428,A -85,B 0,C 180,E1 -21146.121,E2 -21146.121} C_VEL
LIN {X 0,Y 206.352,Z 434.213,A -85,B 0,C 180,E1 -21149.028,E2 -21149.028} C_VEL
LIN {X 0,Y 205.441,Z 439.166,A -85,B 0,C 180,E1 -21151.964,E2 -21151.964} C_VEL
LIN {X 0,Y 204.915,Z 443.378,A -85,B 0,C 180,E1 -21155.275,E2 -21155.275} C_VEL
LIN {X 0,Y 204.511,Z 445.821,A -85,B 0,C 180,E1 -21157.904,E2 -21157.904} C_VEL
LIN {X 0,Y 204.364,Z 447.164,A -85,B 0,C 180,E1 -21159.904,E2 -21159.904} C_VEL
LIN {X 0,Y 204.364,Z 448.111,A -85,B 0,C 180,E1 -21161.91,E2 -21161.91} C_VEL
LIN {X 0,Y 204.593,Z 448.638,A -85,B 0,C 180,E1 -21163.916,E2 -21163.916} C_VEL
LIN {X 0,Y 204.949,Z 448.72,A -85,B 0,C 180,E1 -21166.225,E2 -21166.225} C_VEL
LIN {X 0,Y 205.926,Z 447.765,A -85,B 0,C 180,E1 -21169.957,E2 -21169.957} C_VEL
LIN {X 0,Y 206.746,Z 446.631,A -85,B 0,C 180,E1 -21171.96,E2 -21171.96} C_VEL
LIN {X 0,Y 207.801,Z 444.968,A -85,B 0,C 180,E1 -21174.053,E2 -21174.053} C_VEL
LIN {X 0,Y 209.624,Z 441.857,A -85,B 0,C 180,E1 -21176.912,E2 -21176.912} C_VEL
LIN {X 0,Y 211.977,Z 437.535,A -85,B 0,C 180,E1 -21179.824,E2 -21179.824} C_VEL
LIN {X 0,Y 214.792,Z 431.96,A -85,B 0,C 180,E1 -21182.676,E2 -21182.676} C_VEL
LIN {X 0,Y 218.097,Z 424.938,A -85,B 0,C 180,E1 -21185.453,E2 -21185.453} C_VEL
LIN {X 0,Y 221.822,Z 416.042,A -85,B 0,C 180,E1 -21188.157,E2 -21188.157} C_VEL
LIN {X 0,Y 225.279,Z 406.863,A -85,B 0,C 180,E1 -21190.341,E2 -21190.341} C_VEL
LIN {X 0,Y 228.683,Z 396.676,A -85,B 0,C 180,E1 -21192.242,E2 -21192.242} C_VEL
LIN {X 0,Y 231.759,Z 385.213,A -85,B 0,C 180,E1 -21193.921,E2 -21193.921} C_VEL
LIN {X 0,Y 234.336,Z 373.256,A -85,B 0,C 180,E1 -21195.268,E2 -21195.268} C_VEL
LIN {X 0,Y 236.552,Z 360.63,A -85,B 0,C 180,E1 -21196.274,E2 -21196.274} C_VEL
LIN {X 0,Y 238.037,Z 347.328,A -85,B 0,C 180,E1 -21197.002,E2 -21197.002} C_VEL
LIN {X 0,Y 239.585,Z 321.963,A -85,B 0,C 180,E1 -21197.765,E2 -21197.765} C_VEL
LIN {X 0,Y 240.83,Z 297.862,A -85,B 0,C 180,E1 -21198.454,E2 -21198.454} C_VEL
LIN {X 0,Y 235.016,Z 285.778,A -85,B 0,C 180,E1 -21200.267,E2 -21200.267} C_VEL
LIN {X 0,Y 227.28,Z 273.003,A -85,B 0,C 180,E1 -21202.777,E2 -21202.777} C_VEL
LIN {X 0,Y 220.337,Z 262.731,A -85,B 0,C 180,E1 -21205.239,E2 -21205.239} C_VEL
LIN {X 0,Y 216.725,Z 257.895,A -85,B 0,C 180,E1 -21206.614,E2 -21206.614} C_VEL
LIN {X 0,Y 213.713,Z 253.758,A -85,B 0,C 180,E1 -21207.837,E2 -21207.837} C_VEL
LIN {X 0,Y 211.392,Z 250.961,A -85,B 0,C 180,E1 -21208.805,E2 -21208.805} C_VEL
LIN {X 0,Y 210.258,Z 249.036,A -85,B 0,C 180,E1 -21209.325,E2 -21209.325} C_VEL
LIN {X 0,Y 207.965,Z 246.945,A -85,B 0,C 180,E1 -21210.31,E2 -21210.31} C_VEL
LIN {X 0,Y 206.84,Z 244.396,A -85,B 0,C 180,E1 -21210.901,E2 -21210.901} C_VEL
LIN {X 0,Y 206.732,Z 243.733,A -85,B 0,C 180,E1 -21211.024,E2 -21211.024} C_VEL
LIN {X 0,Y 206.741,Z 243.722,A -85,B 0,C 180,E1 -21215.925,E2 -21215.925} C_VEL
LIN {X 0,Y 206.728,Z 243.722,A -85,B 0,C 180,E1 -21220.125,E2 -21220.125} C_VEL
LIN {X 0,Y 206.844,Z 243.718,A -85,B 0,C 180,E1 -21222.194,E2 -21222.194} C_VEL
LIN {X 0,Y 206.858,Z 243.714,A -85,B 0,C 180,E1 -21226.242,E2 -21226.242} C_VEL
LIN {X 0,Y 207.065,Z 243.685,A -85,B 0,C 180,E1 -21230.229,E2 -21230.229} C_VEL
LIN {X 0,Y 207.042,Z 243.683,A -85,B 0,C 180,E1 -21234.155,E2 -21234.155} C_VEL
LIN {X 0,Y 207.365,Z 243.641,A -85,B 0,C 180,E1 -21238.058,E2 -21238.058} C_VEL
LIN {X 0,Y 207.493,Z 243.635,A -85,B 0,C 180,E1 -21240,E2 -21240} C_VEL
LIN {X 0,Y 207.039,Z 243.684,A -85,B 0,C 180,E1 -21243.893,E2 -21243.893} C_VEL
LIN {X 0,Y 207.106,Z 243.672,A -85,B 0,C 180,E1 -21247.801,E2 -21247.801} C_VEL
LIN {X 0,Y 206.9,Z 243.7,A -85,B 0,C 180,E1 -21251.76,E2 -21251.76} C_VEL
LIN {X 0,Y 206.814,Z 243.716,A -85,B 0,C 180,E1 -21255.775,E2 -21255.775} C_VEL
LIN {X 0,Y 206.706,Z 243.733,A -85,B 0,C 180,E1 -21259.877,E2 -21259.877} C_VEL
LIN {X 0,Y 206.691,Z 243.737,A -85,B 0,C 180,E1 -21264.081,E2 -21264.081} C_VEL
LIN {X 0,Y 206.666,Z 243.738,A -85,B 0,C 180,E1 -21268.43,E2 -21268.43} C_VEL
LIN {X 0,Y 206.685,Z 243.73,A -85,B 0,C 180,E1 -21272.96,E2 -21272.96} C_VEL
LIN {X 0,Y 206.721,Z 243.763,A -85,B 0,C 180,E1 -21275.137,E2 -21275.137} C_VEL
LIN {X 0,Y 208.674,Z 249.99,A -85,B 0,C 180,E1 -21279.785,E2 -21279.785} C_VEL
LIN {X 0,Y 209.209,Z 251.564,A -85,B 0,C 180,E1 -21280.845,E2 -21280.845} C_VEL
LIN {X 0,Y 211.853,Z 255.991,A -85,B 0,C 180,E1 -21282.054,E2 -21282.054} C_VEL
LIN {X 0,Y 213.523,Z 258.223,A -85,B 0,C 180,E1 -21282.755,E2 -21282.755} C_VEL
LIN {X 0,Y 217.571,Z 264.672,A -85,B 0,C 180,E1 -21284.421,E2 -21284.421} C_VEL
LIN {X 0,Y 219.022,Z 267.073,A -85,B 0,C 180,E1 -21284.993,E2 -21284.993} C_VEL
LIN {X 0,Y 220.251,Z 269.439,A -85,B 0,C 180,E1 -21285.482,E2 -21285.482} C_VEL
LIN {X 0,Y 221.106,Z 273.679,A -85,B 0,C 180,E1 -21285.941,E2 -21285.941} C_VEL
LIN {X 0,Y 222.056,Z 282.849,A -85,B 0,C 180,E1 -21286.655,E2 -21286.655} C_VEL
LIN {X 0,Y 223.239,Z 286.226,A -85,B 0,C 180,E1 -21287.146,E2 -21287.146} C_VEL
LIN {X 0,Y 228.013,Z 296.143,A -85,B 0,C 180,E1 -21288.871,E2 -21288.871} C_VEL
LIN {X 0,Y 232.901,Z 307.547,A -85,B 0,C 180,E1 -21290.566,E2 -21290.566} C_VEL
LIN {X 0,Y 234.519,Z 319.939,A -85,B 0,C 180,E1 -21291.458,E2 -21291.458} C_VEL
LIN {X 0,Y 232.012,Z 362.571,A -85,B 0,C 180,E1 -21292.712,E2 -21292.712} C_VEL
LIN {X 0,Y 230.328,Z 376.304,A -85,B 0,C 180,E1 -21293.419,E2 -21293.419} C_VEL
LIN {X 0,Y 227.792,Z 389.228,A -85,B 0,C 180,E1 -21294.384,E2 -21294.384} C_VEL
LIN {X 0,Y 224.535,Z 401.767,A -85,B 0,C 180,E1 -21295.708,E2 -21295.708} C_VEL
LIN {X 0,Y 221.164,Z 412.943,A -85,B 0,C 180,E1 -21297.301,E2 -21297.301} C_VEL
LIN {X 0,Y 217.487,Z 423.046,A -85,B 0,C 180,E1 -21299.136,E2 -21299.136} C_VEL
LIN {X 0,Y 213.485,Z 432.978,A -85,B 0,C 180,E1 -21301.487,E2 -21301.487} C_VEL
LIN {X 0,Y 209.52,Z 441.755,A -85,B 0,C 180,E1 -21304.146,E2 -21304.146} C_VEL
LIN {X 0,Y 206.114,Z 449.01,A -85,B 0,C 180,E1 -21307.02,E2 -21307.02} C_VEL
LIN {X 0,Y 203.463,Z 454.469,A -85,B 0,C 180,E1 -21309.791,E2 -21309.791} C_VEL
LIN {X 0,Y 201.149,Z 458.958,A -85,B 0,C 180,E1 -21312.721,E2 -21312.721} C_VEL
LIN {X 0,Y 199.336,Z 462.393,A -85,B 0,C 180,E1 -21315.709,E2 -21315.709} C_VEL
LIN {X 0,Y 197.948,Z 465.456,A -85,B 0,C 180,E1 -21319.772,E2 -21319.772} C_VEL
LIN {X 0,Y 197.53,Z 466.403,A -85,B 0,C 180,E1 -21321.815,E2 -21321.815} C_VEL
LIN {X 0,Y 197.341,Z 467.09,A -85,B 0,C 180,E1 -21325.695,E2 -21325.695} C_VEL
LIN {X 0,Y 197.462,Z 466.824,A -85,B 0,C 180,E1 -21327.957,E2 -21327.957} C_VEL
LIN {X 0,Y 197.609,Z 466.179,A -85,B 0,C 180,E1 -21329.996,E2 -21329.996} C_VEL
LIN {X 0,Y 197.497,Z 465.11,A -85,B 0,C 180,E1 -21332.035,E2 -21332.035} C_VEL
LIN {X 0,Y 197.373,Z 463.268,A -85,B 0,C 180,E1 -21334.425,E2 -21334.425} C_VEL
LIN {X 0,Y 197.505,Z 460.466,A -85,B 0,C 180,E1 -21337.15,E2 -21337.15} C_VEL
LIN {X 0,Y 197.907,Z 456.27,A -85,B 0,C 180,E1 -21340.223,E2 -21340.223} C_VEL
LIN {X 0,Y 198.844,Z 449.843,A -85,B 0,C 180,E1 -21343.797,E2 -21343.797} C_VEL
LIN {X 0,Y 200.332,Z 442.845,A -85,B 0,C 180,E1 -21346.818,E2 -21346.818} C_VEL
LIN {X 0,Y 202.002,Z 434.482,A -85,B 0,C 180,E1 -21349.677,E2 -21349.677} C_VEL
LIN {X 0,Y 204.175,Z 425.007,A -85,B 0,C 180,E1 -21352.243,E2 -21352.243} C_VEL
LIN {X 0,Y 206.196,Z 415.061,A -85,B 0,C 180,E1 -21354.404,E2 -21354.404} C_VEL
LIN {X 0,Y 208.359,Z 404.087,A -85,B 0,C 180,E1 -21356.27,E2 -21356.27} C_VEL
LIN {X 0,Y 210.293,Z 392.759,A -85,B 0,C 180,E1 -21357.754,E2 -21357.754} C_VEL
LIN {X 0,Y 211.901,Z 381.431,A -85,B 0,C 180,E1 -21358.873,E2 -21358.873} C_VEL
LIN {X 0,Y 213.324,Z 367.846,A -85,B 0,C 180,E1 -21359.814,E2 -21359.814} C_VEL
LIN {X 0,Y 214.147,Z 352.976,A -85,B 0,C 180,E1 -21360.406,E2 -21360.406} C_VEL
LIN {X 0,Y 215.524,Z 311.6,A -85,B 0,C 180,E1 -21361.746,E2 -21361.746} C_VEL
LIN {X 0,Y 212.225,Z 280.032,A -85,B 0,C 180,E1 -21363.389,E2 -21363.389} C_VEL
LIN {X 0,Y 208.386,Z 269.365,A -85,B 0,C 180,E1 -21364.377,E2 -21364.377} C_VEL
LIN {X 0,Y 202.816,Z 256.244,A -85,B 0,C 180,E1 -21365.8,E2 -21365.8} C_VEL
LIN {X 0,Y 201.772,Z 253.513,A -85,B 0,C 180,E1 -21366.141,E2 -21366.141} C_VEL
LIN {X 0,Y 200.17,Z 246.644,A -85,B 0,C 180,E1 -21369.428,E2 -21369.428} C_VEL
LIN {X 0,Y 199.642,Z 244.618,A -85,B 0,C 180,E1 -21370.532,E2 -21370.532} C_VEL
LIN {X 0,Y 199.596,Z 244.621,A -85,B 0,C 180,E1 -21375.233,E2 -21375.233} C_VEL
LIN {X 0,Y 199.634,Z 244.618,A -85,B 0,C 180,E1 -21378.019,E2 -21378.019} C_VEL
LIN {X 0,Y 199.658,Z 244.615,A -85,B 0,C 180,E1 -21380.738,E2 -21380.738} C_VEL
LIN {X 0,Y 199.587,Z 244.623,A -85,B 0,C 180,E1 -21385.709,E2 -21385.709} C_VEL
LIN {X 0,Y 199.667,Z 244.614,A -85,B 0,C 180,E1 -21388.131,E2 -21388.131} C_VEL
LIN {X 0,Y 199.661,Z 244.613,A -85,B 0,C 180,E1 -21392.768,E2 -21392.768} C_VEL
LIN {X 0,Y 199.728,Z 244.604,A -85,B 0,C 180,E1 -21397.228,E2 -21397.228} C_VEL
LIN {X 0,Y 199.808,Z 244.593,A -85,B 0,C 180,E1 -21401.719,E2 -21401.719} C_VEL
LIN {X 0,Y 199.794,Z 244.592,A -85,B 0,C 180,E1 -21405.745,E2 -21405.745} C_VEL
LIN {X 0,Y 199.991,Z 244.572,A -85,B 0,C 180,E1 -21409.88,E2 -21409.88} C_VEL
LIN {X 0,Y 199.987,Z 244.57,A -85,B 0,C 180,E1 -21413.948,E2 -21413.948} C_VEL
LIN {X 0,Y 200.283,Z 244.531,A -85,B 0,C 180,E1 -21417.989,E2 -21417.989} C_VEL
LIN {X 0,Y 200.435,Z 244.498,A -85,B 0,C 180,E1 -21420,E2 -21420} C_VEL
LIN {X 0,Y 199.978,Z 244.555,A -85,B 0,C 180,E1 -21424.031,E2 -21424.031} C_VEL
LIN {X 0,Y 200.042,Z 244.564,A -85,B 0,C 180,E1 -21428.079,E2 -21428.079} C_VEL
LIN {X 0,Y 199.827,Z 244.575,A -85,B 0,C 180,E1 -21432.183,E2 -21432.183} C_VEL
LIN {X 0,Y 199.716,Z 244.588,A -85,B 0,C 180,E1 -21436.351,E2 -21436.351} C_VEL
LIN {X 0,Y 199.615,Z 244.621,A -85,B 0,C 180,E1 -21440.615,E2 -21440.615} C_VEL
LIN {X 0,Y 199.632,Z 244.618,A -85,B 0,C 180,E1 -21444.99,E2 -21444.99} C_VEL
LIN {X 0,Y 199.638,Z 244.612,A -85,B 0,C 180,E1 -21449.529,E2 -21449.529} C_VEL
LIN {X 0,Y 199.646,Z 244.617,A -85,B 0,C 180,E1 -21452.36,E2 -21452.36} C_VEL
LIN {X 0,Y 199.623,Z 244.619,A -85,B 0,C 180,E1 -21456.764,E2 -21456.764} C_VEL
LIN {X 0,Y 199.657,Z 244.606,A -85,B 0,C 180,E1 -21459.317,E2 -21459.317} C_VEL
LIN {X 0,Y 199.627,Z 244.616,A -85,B 0,C 180,E1 -21462.338,E2 -21462.338} C_VEL
LIN {X 0,Y 199.579,Z 244.605,A -85,B 0,C 180,E1 -21465.239,E2 -21465.239} C_VEL
LIN {X 0,Y 199.56,Z 244.618,A -85,B 0,C 180,E1 -21468.01,E2 -21468.01} C_VEL
LIN {X 0,Y 199.585,Z 244.618,A -85,B 0,C 180,E1 -21470.777,E2 -21470.777} C_VEL
LIN {X 0,Y 199.6,Z 244.621,A -85,B 0,C 180,E1 -21475.719,E2 -21475.719} C_VEL
LIN {X 0,Y 199.682,Z 244.612,A -85,B 0,C 180,E1 -21478.142,E2 -21478.142} C_VEL
LIN {X 0,Y 199.676,Z 244.611,A -85,B 0,C 180,E1 -21482.777,E2 -21482.777} C_VEL
LIN {X 0,Y 199.672,Z 244.608,A -85,B 0,C 180,E1 -21484.883,E2 -21484.883} C_VEL
LIN {X 0,Y 200.729,Z 247.533,A -85,B 0,C 180,E1 -21485.207,E2 -21485.207} C_VEL
LIN {X 0,Y 205.101,Z 255.199,A -85,B 0,C 180,E1 -21486.261,E2 -21486.261} C_VEL
LIN {X 0,Y 213.137,Z 271.84,A -85,B 0,C 180,E1 -21488.158,E2 -21488.158} C_VEL
LIN {X 0,Y 216.224,Z 279.35,A -85,B 0,C 180,E1 -21488.883,E2 -21488.883} C_VEL
LIN {X 0,Y 216.724,Z 281.692,A -85,B 0,C 180,E1 -21489.039,E2 -21489.039} C_VEL
LIN {X 0,Y 214.087,Z 345.485,A -85,B 0,C 180,E1 -21491.09,E2 -21491.09} C_VEL
LIN {X 0,Y 213.02,Z 357.86,A -85,B 0,C 180,E1 -21491.802,E2 -21491.802} C_VEL
LIN {X 0,Y 211.916,Z 368.936,A -85,B 0,C 180,E1 -21492.764,E2 -21492.764} C_VEL
LIN {X 0,Y 210.348,Z 381.522,A -85,B 0,C 180,E1 -21494.254,E2 -21494.254} C_VEL
LIN {X 0,Y 208.169,Z 393.366,A -85,B 0,C 180,E1 -21496.086,E2 -21496.086} C_VEL
LIN {X 0,Y 206.079,Z 403.914,A -85,B 0,C 180,E1 -21498.198,E2 -21498.198} C_VEL
LIN {X 0,Y 203.94,Z 413.444,A -85,B 0,C 180,E1 -21500.584,E2 -21500.584} C_VEL
LIN {X 0,Y 201.991,Z 422.577,A -85,B 0,C 180,E1 -21503.512,E2 -21503.512} C_VEL
LIN {X 0,Y 200.265,Z 429.954,A -85,B 0,C 180,E1 -21506.483,E2 -21506.483} C_VEL
LIN {X 0,Y 198.943,Z 436.724,A -85,B 0,C 180,E1 -21510.004,E2 -21510.004} C_VEL
LIN {X 0,Y 198.159,Z 441.201,A -85,B 0,C 180,E1 -21513.053,E2 -21513.053} C_VEL
LIN {X 0,Y 197.676,Z 444.611,A -85,B 0,C 180,E1 -21516.126,E2 -21516.126} C_VEL
LIN {X 0,Y 197.395,Z 446.321,A -85,B 0,C 180,E1 -21518.191,E2 -21518.191} C_VEL
LIN {X 0,Y 197.253,Z 447.627,A -85,B 0,C 180,E1 -21520.265,E2 -21520.265} C_VEL
LIN {X 0,Y 197.301,Z 448.533,A -85,B 0,C 180,E1 -21522.343,E2 -21522.343} C_VEL
LIN {X 0,Y 197.55,Z 448.991,A -85,B 0,C 180,E1 -21524.423,E2 -21524.423} C_VEL
LIN {X 0,Y 197.914,Z 449.054,A -85,B 0,C 180,E1 -21526.506,E2 -21526.506} C_VEL
LIN {X 0,Y 198.383,Z 448.728,A -85,B 0,C 180,E1 -21528.595,E2 -21528.595} C_VEL
LIN {X 0,Y 199.068,Z 447.992,A -85,B 0,C 180,E1 -21530.676,E2 -21530.676} C_VEL
LIN {X 0,Y 200.965,Z 445.36,A -85,B 0,C 180,E1 -21534.597,E2 -21534.597} C_VEL
LIN {X 0,Y 203.11,Z 441.903,A -85,B 0,C 180,E1 -21537.849,E2 -21537.849} C_VEL
LIN {X 0,Y 205.63,Z 437.494,A -85,B 0,C 180,E1 -21540.843,E2 -21540.843} C_VEL
LIN {X 0,Y 208.664,Z 431.825,A -85,B 0,C 180,E1 -21543.762,E2 -21543.762} C_VEL
LIN {X 0,Y 212.184,Z 424.653,A -85,B 0,C 180,E1 -21546.598,E2 -21546.598} C_VEL
LIN {X 0,Y 216.106,Z 415.616,A -85,B 0,C 180,E1 -21549.358,E2 -21549.358} C_VEL
LIN {X 0,Y 219.765,Z 406.284,A -85,B 0,C 180,E1 -21551.573,E2 -21551.573} C_VEL
LIN {X 0,Y 223.264,Z 396.009,A -85,B 0,C 180,E1 -21553.471,E2 -21553.471} C_VEL
LIN {X 0,Y 226.489,Z 384.227,A -85,B 0,C 180,E1 -21555.187,E2 -21555.187} C_VEL
LIN {X 0,Y 229.039,Z 372.749,A -85,B 0,C 180,E1 -21556.462,E2 -21556.462} C_VEL
LIN {X 0,Y 231.279,Z 360.013,A -85,B 0,C 180,E1 -21557.462,E2 -21557.462} C_VEL
LIN {X 0,Y 232.74,Z 347.259,A -85,B 0,C 180,E1 -21558.152,E2 -21558.152} C_VEL
LIN {X 0,Y 235.092,Z 307.582,A -85,B 0,C 180,E1 -21559.338,E2 -21559.338} C_VEL
LIN {X 0,Y 235.464,Z 300.142,A -85,B 0,C 180,E1 -21559.561,E2 -21559.561} C_VEL
LIN {X 0,Y 230.475,Z 289.845,A -85,B 0,C 180,E1 -21561.199,E2 -21561.199} C_VEL
LIN {X 0,Y 223.19,Z 277.645,A -85,B 0,C 180,E1 -21563.686,E2 -21563.686} C_VEL
LIN {X 0,Y 216.701,Z 267.956,A -85,B 0,C 180,E1 -21566.104,E2 -21566.104} C_VEL
LIN {X 0,Y 212.959,Z 262.869,A -85,B 0,C 180,E1 -21567.604,E2 -21567.604} C_VEL
LIN {X 0,Y 210.434,Z 259.395,A -85,B 0,C 180,E1 -21568.679,E2 -21568.679} C_VEL
LIN {X 0,Y 207.896,Z 255.961,A -85,B 0,C 180,E1 -21569.811,E2 -21569.811} C_VEL
LIN {X 0,Y 206.983,Z 254.839,A -85,B 0,C 180,E1 -21570.225,E2 -21570.225} C_VEL
LIN {X 0,Y 204.531,Z 251.912,A -85,B 0,C 180,E1 -21571.375,E2 -21571.375} C_VEL
LIN {X 0,Y 203.531,Z 250.049,A -85,B 0,C 180,E1 -21571.904,E2 -21571.904} C_VEL
LIN {X 0,Y 201.043,Z 247.969,A -85,B 0,C 180,E1 -21573.111,E2 -21573.111} C_VEL
LIN {X 0,Y 199.807,Z 245.339,A -85,B 0,C 180,E1 -21573.846,E2 -21573.846} C_VEL
LIN {X 0,Y 199.674,Z 244.61,A -85,B 0,C 180,E1 -21574.038,E2 -21574.038} C_VEL
LIN {X 0,Y 199.706,Z 244.599,A -85,B 0,C 180,E1 -21577.225,E2 -21577.225} C_VEL
LIN {X 0,Y 199.75,Z 244.597,A -85,B 0,C 180,E1 -21581.795,E2 -21581.795} C_VEL
LIN {X 0,Y 199.799,Z 244.588,A -85,B 0,C 180,E1 -21585.745,E2 -21585.745} C_VEL
LIN {X 0,Y 200.018,Z 244.56,A -85,B 0,C 180,E1 -21589.881,E2 -21589.881} C_VEL
LIN {X 0,Y 200.004,Z 244.559,A -85,B 0,C 180,E1 -21593.949,E2 -21593.949} C_VEL
LIN {X 0,Y 200.305,Z 244.52,A -85,B 0,C 180,E1 -21597.989,E2 -21597.989} C_VEL
LIN {X 0,Y 200.458,Z 244.511,A -85,B 0,C 180,E1 -21600,E2 -21600} C_VEL
LIN {X 0,Y 199.985,Z 244.563,A -85,B 0,C 180,E1 -21604.03,E2 -21604.03} C_VEL
LIN {X 0,Y 200.055,Z 244.55,A -85,B 0,C 180,E1 -21608.078,E2 -21608.078} C_VEL
LIN {X 0,Y 199.852,Z 244.576,A -85,B 0,C 180,E1 -21612.181,E2 -21612.181} C_VEL
LIN {X 0,Y 199.747,Z 244.591,A -85,B 0,C 180,E1 -21616.348,E2 -21616.348} C_VEL
LIN {X 0,Y 199.638,Z 244.606,A -85,B 0,C 180,E1 -21620.612,E2 -21620.612} C_VEL
LIN {X 0,Y 199.612,Z 244.61,A -85,B 0,C 180,E1 -21624.992,E2 -21624.992} C_VEL
LIN {X 0,Y 199.592,Z 244.612,A -85,B 0,C 180,E1 -21629.536,E2 -21629.536} C_VEL
LIN {X 0,Y 199.676,Z 244.711,A -85,B 0,C 180,E1 -21632.681,E2 -21632.681} C_VEL
LIN {X 0,Y 201.115,Z 249.279,A -85,B 0,C 180,E1 -21636.513,E2 -21636.513} C_VEL
LIN {X 0,Y 201.832,Z 251.157,A -85,B 0,C 180,E1 -21637.858,E2 -21637.858} C_VEL
LIN {X 0,Y 204.849,Z 255.831,A -85,B 0,C 180,E1 -21639.408,E2 -21639.408} C_VEL
LIN {X 0,Y 206.446,Z 257.925,A -85,B 0,C 180,E1 -21640.164,E2 -21640.164} C_VEL
LIN {X 0,Y 209.555,Z 262.675,A -85,B 0,C 180,E1 -21641.604,E2 -21641.604} C_VEL
LIN {X 0,Y 214.474,Z 270.641,A -85,B 0,C 180,E1 -21643.732,E2 -21643.732} C_VEL
LIN {X 0,Y 219.508,Z 279.26,A -85,B 0,C 180,E1 -21645.741,E2 -21645.741} C_VEL
LIN {X 0,Y 223.239,Z 286.226,A -85,B 0,C 180,E1 -21647.146,E2 -21647.146} C_VEL
LIN {X 0,Y 225.247,Z 290.905,A -85,B 0,C 180,E1 -21647.911,E2 -21647.911} C_VEL
LIN {X 0,Y 226.56,Z 296.218,A -85,B 0,C 180,E1 -21648.499,E2 -21648.499} C_VEL
LIN {X 0,Y 227.142,Z 299.944,A -85,B 0,C 180,E1 -21648.817,E2 -21648.817} C_VEL
LIN {X 0,Y 228.678,Z 315.581,A -85,B 0,C 180,E1 -21649.892,E2 -21649.892} C_VEL
LIN {X 0,Y 229.327,Z 321.16,A -85,B 0,C 180,E1 -21650.292,E2 -21650.292} C_VEL
LIN {X 0,Y 226.737,Z 362.709,A -85,B 0,C 180,E1 -21651.534,E2 -21651.534} C_VEL
LIN {X 0,Y 224.952,Z 376.433,A -85,B 0,C 180,E1 -21652.255,E2 -21652.255} C_VEL
LIN {X 0,Y 222.343,Z 389.196,A -85,B 0,C 180,E1 -21653.231,E2 -21653.231} C_VEL
LIN {X 0,Y 219.212,Z 400.886,A -85,B 0,C 180,E1 -21654.472,E2 -21654.472} C_VEL
LIN {X 0,Y 215.689,Z 412.163,A -85,B 0,C 180,E1 -21656.082,E2 -21656.082} C_VEL
LIN {X 0,Y 211.832,Z 422.368,A -85,B 0,C 180,E1 -21657.937,E2 -21657.937} C_VEL
LIN {X 0,Y 208.01,Z 431.552,A -85,B 0,C 180,E1 -21660.108,E2 -21660.108} C_VEL
LIN {X 0,Y 203.801,Z 440.512,A -85,B 0,C 180,E1 -21662.81,E2 -21662.81} C_VEL
LIN {X 0,Y 200.036,Z 448.144,A -85,B 0,C 180,E1 -21665.813,E2 -21665.813} C_VEL
LIN {X 0,Y 196.808,Z 454.402,A -85,B 0,C 180,E1 -21669.076,E2 -21669.076} C_VEL
LIN {X 0,Y 194.362,Z 458.831,A -85,B 0,C 180,E1 -21672.098,E2 -21672.098} C_VEL
LIN {X 0,Y 192.425,Z 462.208,A -85,B 0,C 180,E1 -21675.185,E2 -21675.185} C_VEL
LIN {X 0,Y 190.948,Z 465.218,A -85,B 0,C 180,E1 -21679.392,E2 -21679.392} C_VEL
LIN {X 0,Y 190.487,Z 466.137,A -85,B 0,C 180,E1 -21681.51,E2 -21681.51} C_VEL
LIN {X 0,Y 190.277,Z 466.738,A -85,B 0,C 180,E1 -21685.76,E2 -21685.76} C_VEL
LIN {X 0,Y 190.377,Z 466.459,A -85,B 0,C 180,E1 -21687.881,E2 -21687.881} C_VEL
LIN {X 0,Y 190.52,Z 465.789,A -85,B 0,C 180,E1 -21689.996,E2 -21689.996} C_VEL
LIN {X 0,Y 190.411,Z 464.671,A -85,B 0,C 180,E1 -21692.111,E2 -21692.111} C_VEL
LIN {X 0,Y 190.302,Z 463.013,A -85,B 0,C 180,E1 -21694.339,E2 -21694.339} C_VEL
LIN {X 0,Y 190.449,Z 459.941,A -85,B 0,C 180,E1 -21697.416,E2 -21697.416} C_VEL
LIN {X 0,Y 190.865,Z 455.682,A -85,B 0,C 180,E1 -21700.604,E2 -21700.604} C_VEL
LIN {X 0,Y 191.927,Z 449.192,A -85,B 0,C 180,E1 -21704.305,E2 -21704.305} C_VEL
LIN {X 0,Y 193.462,Z 442.092,A -85,B 0,C 180,E1 -21707.434,E2 -21707.434} C_VEL
LIN {X 0,Y 194.968,Z 435.259,A -85,B 0,C 180,E1 -21709.872,E2 -21709.872} C_VEL
LIN {X 0,Y 197.123,Z 426.023,A -85,B 0,C 180,E1 -21712.53,E2 -21712.53} C_VEL
LIN {X 0,Y 199.434,Z 415.154,A -85,B 0,C 180,E1 -21715.01,E2 -21715.01} C_VEL
LIN {X 0,Y 201.692,Z 404.324,A -85,B 0,C 180,E1 -21716.928,E2 -21716.928} C_VEL
LIN {X 0,Y 203.678,Z 393.138,A -85,B 0,C 180,E1 -21718.457,E2 -21718.457} C_VEL
LIN {X 0,Y 205.358,Z 382.03,A -85,B 0,C 180,E1 -21719.603,E2 -21719.603} C_VEL
LIN {X 0,Y 206.818,Z 368.871,A -85,B 0,C 180,E1 -21720.567,E2 -21720.567} C_VEL
LIN {X 0,Y 207.637,Z 355.908,A -85,B 0,C 180,E1 -21721.153,E2 -21721.153} C_VEL
LIN {X 0,Y 209.257,Z 313.008,A -85,B 0,C 180,E1 -21722.562,E2 -21722.562} C_VEL
LIN {X 0,Y 206.137,Z 282.006,A -85,B 0,C 180,E1 -21724.231,E2 -21724.231} C_VEL
LIN {X 0,Y 200.667,Z 267.457,A -85,B 0,C 180,E1 -21725.706,E2 -21725.706} C_VEL
LIN {X 0,Y 195.451,Z 255.752,A -85,B 0,C 180,E1 -21727.116,E2 -21727.116} C_VEL
LIN {X 0,Y 194.489,Z 253.203,A -85,B 0,C 180,E1 -21727.43,E2 -21727.43} C_VEL
LIN {X 0,Y 192.542,Z 245.502,A -85,B 0,C 180,E1 -21731.41,E2 -21731.41} C_VEL
LIN {X 0,Y 192.543,Z 245.502,A -85,B 0,C 180,E1 -21736.876,E2 -21736.876} C_VEL
LIN {X 0,Y 192.576,Z 245.5,A -85,B 0,C 180,E1 -21741.654,E2 -21741.654} C_VEL
LIN {X 0,Y 192.583,Z 245.495,A -85,B 0,C 180,E1 -21747.055,E2 -21747.055} C_VEL
LIN {X 0,Y 192.638,Z 245.49,A -85,B 0,C 180,E1 -21751.688,E2 -21751.688} C_VEL
LIN {X 0,Y 192.687,Z 245.481,A -85,B 0,C 180,E1 -21756.346,E2 -21756.346} C_VEL
LIN {X 0,Y 192.753,Z 245.472,A -85,B 0,C 180,E1 -21761.411,E2 -21761.411} C_VEL
LIN {X 0,Y 192.724,Z 245.476,A -85,B 0,C 180,E1 -21765.211,E2 -21765.211} C_VEL
LIN {X 0,Y 192.915,Z 245.455,A -85,B 0,C 180,E1 -21769.565,E2 -21769.565} C_VEL
LIN {X 0,Y 192.95,Z 245.446,A -85,B 0,C 180,E1 -21773.727,E2 -21773.727} C_VEL
LIN {X 0,Y 193.225,Z 245.41,A -85,B 0,C 180,E1 -21777.916,E2 -21777.916} C_VEL
LIN {X 0,Y 193.4,Z 245.372,A -85,B 0,C 180,E1 -21780,E2 -21780} C_VEL
LIN {X 0,Y 192.924,Z 245.434,A -85,B 0,C 180,E1 -21784.178,E2 -21784.178} C_VEL
LIN {X 0,Y 192.993,Z 245.443,A -85,B 0,C 180,E1 -21788.376,E2 -21788.376} C_VEL
LIN {X 0,Y 192.748,Z 245.451,A -85,B 0,C 180,E1 -21792.637,E2 -21792.637} C_VEL
LIN {X 0,Y 192.665,Z 245.48,A -85,B 0,C 180,E1 -21798.511,E2 -21798.511} C_VEL
LIN {X 0,Y 192.611,Z 245.486,A -85,B 0,C 180,E1 -21804.211,E2 -21804.211} C_VEL
LIN {X 0,Y 192.618,Z 245.485,A -85,B 0,C 180,E1 -21808.893,E2 -21808.893} C_VEL
LIN {X 0,Y 192.573,Z 245.494,A -85,B 0,C 180,E1 -21813.191,E2 -21813.191} C_VEL
LIN {X 0,Y 192.577,Z 245.492,A -85,B 0,C 180,E1 -21818.346,E2 -21818.346} C_VEL
LIN {X 0,Y 192.544,Z 245.495,A -85,B 0,C 180,E1 -21823.124,E2 -21823.124} C_VEL
LIN {X 0,Y 192.498,Z 245.488,A -85,B 0,C 180,E1 -21826.903,E2 -21826.903} C_VEL
LIN {X 0,Y 192.53,Z 245.492,A -85,B 0,C 180,E1 -21831.653,E2 -21831.653} C_VEL
LIN {X 0,Y 192.585,Z 245.493,A -85,B 0,C 180,E1 -21836.82,E2 -21836.82} C_VEL
LIN {X 0,Y 192.652,Z 245.488,A -85,B 0,C 180,E1 -21841.697,E2 -21841.697} C_VEL
LIN {X 0,Y 192.648,Z 245.487,A -85,B 0,C 180,E1 -21843.609,E2 -21843.609} C_VEL
LIN {X 0,Y 193.765,Z 248.524,A -85,B 0,C 180,E1 -21843.982,E2 -21843.982} C_VEL
LIN {X 0,Y 200.488,Z 260.552,A -85,B 0,C 180,E1 -21845.703,E2 -21845.703} C_VEL
LIN {X 0,Y 208.192,Z 276.803,A -85,B 0,C 180,E1 -21847.607,E2 -21847.607} C_VEL
LIN {X 0,Y 210.338,Z 282.232,A -85,B 0,C 180,E1 -21848.141,E2 -21848.141} C_VEL
LIN {X 0,Y 207.733,Z 345.384,A -85,B 0,C 180,E1 -21850.231,E2 -21850.231} C_VEL
LIN {X 0,Y 206.611,Z 357.908,A -85,B 0,C 180,E1 -21850.959,E2 -21850.959} C_VEL
LIN {X 0,Y 205.48,Z 369.047,A -85,B 0,C 180,E1 -21851.949,E2 -21851.949} C_VEL
LIN {X 0,Y 203.839,Z 381.678,A -85,B 0,C 180,E1 -21853.48,E2 -21853.48} C_VEL
LIN {X 0,Y 201.575,Z 393.567,A -85,B 0,C 180,E1 -21855.364,E2 -21855.364} C_VEL
LIN {X 0,Y 199.394,Z 404.136,A -85,B 0,C 180,E1 -21857.538,E2 -21857.538} C_VEL
LIN {X 0,Y 197.37,Z 412.794,A -85,B 0,C 180,E1 -21859.749,E2 -21859.749} C_VEL
LIN {X 0,Y 195.586,Z 420.741,A -85,B 0,C 180,E1 -21862.261,E2 -21862.261} C_VEL
LIN {X 0,Y 193.675,Z 428.556,A -85,B 0,C 180,E1 -21865.321,E2 -21865.321} C_VEL
LIN {X 0,Y 192.516,Z 433.859,A -85,B 0,C 180,E1 -21867.912,E2 -21867.912} C_VEL
LIN {X 0,Y 191.51,Z 439.031,A -85,B 0,C 180,E1 -21871.055,E2 -21871.055} C_VEL
LIN {X 0,Y 190.896,Z 443.055,A -85,B 0,C 180,E1 -21874.226,E2 -21874.226} C_VEL
LIN {X 0,Y 190.532,Z 445.147,A -85,B 0,C 180,E1 -21876.357,E2 -21876.357} C_VEL
LIN {X 0,Y 190.275,Z 446.818,A -85,B 0,C 180,E1 -21878.499,E2 -21878.499} C_VEL
LIN {X 0,Y 190.166,Z 448.088,A -85,B 0,C 180,E1 -21880.652,E2 -21880.652} C_VEL
LIN {X 0,Y 190.254,Z 448.928,A -85,B 0,C 180,E1 -21882.808,E2 -21882.808} C_VEL
LIN {X 0,Y 190.862,Z 449.39,A -85,B 0,C 180,E1 -21886.786,E2 -21886.786} C_VEL
LIN {X 0,Y 191.471,Z 449.007,A -85,B 0,C 180,E1 -21889.292,E2 -21889.292} C_VEL
LIN {X 0,Y 192.244,Z 448.198,A -85,B 0,C 180,E1 -21891.445,E2 -21891.445} C_VEL
LIN {X 0,Y 194.15,Z 445.753,A -85,B 0,C 180,E1 -21895.18,E2 -21895.18} C_VEL
LIN {X 0,Y 196.65,Z 441.949,A -85,B 0,C 180,E1 -21898.848,E2 -21898.848} C_VEL
LIN {X 0,Y 199.908,Z 436.515,A -85,B 0,C 180,E1 -21902.461,E2 -21902.461} C_VEL
LIN {X 0,Y 203.799,Z 429.411,A -85,B 0,C 180,E1 -21905.891,E2 -21905.891} C_VEL
LIN {X 0,Y 207.218,Z 422.567,A -85,B 0,C 180,E1 -21908.425,E2 -21908.425} C_VEL
LIN {X 0,Y 210.484,Z 415.191,A -85,B 0,C 180,E1 -21910.625,E2 -21910.625} C_VEL
LIN {X 0,Y 214.342,Z 405.639,A -85,B 0,C 180,E1 -21912.872,E2 -21912.872} C_VEL
LIN {X 0,Y 218.15,Z 394.699,A -85,B 0,C 180,E1 -21914.865,E2 -21914.865} C_VEL
LIN {X 0,Y 221.428,Z 382.893,A -85,B 0,C 180,E1 -21916.554,E2 -21916.554} C_VEL
LIN {X 0,Y 223.854,Z 372.183,A -85,B 0,C 180,E1 -21917.71,E2 -21917.71} C_VEL
LIN {X 0,Y 226.22,Z 358.696,A -85,B 0,C 180,E1 -21918.751,E2 -21918.751} C_VEL
LIN {X 0,Y 227.624,Z 346.364,A -85,B 0,C 180,E1 -21919.394,E2 -21919.394} C_VEL
LIN {X 0,Y 230.197,Z 302.553,A -85,B 0,C 180,E1 -21920.715,E2 -21920.715} C_VEL
LIN {X 0,Y 226.168,Z 294.224,A -85,B 0,C 180,E1 -21922.11,E2 -21922.11} C_VEL
LIN {X 0,Y 219.268,Z 282.485,A -85,B 0,C 180,E1 -21924.588,E2 -21924.588} C_VEL
LIN {X 0,Y 213.151,Z 273.182,A -85,B 0,C 180,E1 -21926.988,E2 -21926.988} C_VEL
LIN {X 0,Y 207.427,Z 265.189,A -85,B 0,C 180,E1 -21929.454,E2 -21929.454} C_VEL
LIN {X 0,Y 204.11,Z 260.791,A -85,B 0,C 180,E1 -21931.004,E2 -21931.004} C_VEL
LIN {X 0,Y 201.381,Z 257.219,A -85,B 0,C 180,E1 -21932.365,E2 -21932.365} C_VEL
LIN {X 0,Y 200.584,Z 256.103,A -85,B 0,C 180,E1 -21932.784,E2 -21932.784} C_VEL
LIN {X 0,Y 198.086,Z 253.48,A -85,B 0,C 180,E1 -21934.097,E2 -21934.097} C_VEL
LIN {X 0,Y 196.728,Z 251.077,A -85,B 0,C 180,E1 -21934.916,E2 -21934.916} C_VEL
LIN {X 0,Y 194.267,Z 249.143,A -85,B 0,C 180,E1 -21936.303,E2 -21936.303} C_VEL
LIN {X 0,Y 192.982,Z 246.861,A -85,B 0,C 180,E1 -21937.165,E2 -21937.165} C_VEL
LIN {X 0,Y 192.655,Z 245.479,A -85,B 0,C 180,E1 -21937.478,E2 -21937.478} C_VEL
LIN {X 0,Y 192.717,Z 245.476,A -85,B 0,C 180,E1 -21943.037,E2 -21943.037} C_VEL
LIN {X 0,Y 192.779,Z 245.47,A -85,B 0,C 180,E1 -21947.365,E2 -21947.365} C_VEL
LIN {X 0,Y 193.019,Z 245.442,A -85,B 0,C 180,E1 -21951.625,E2 -21951.625} C_VEL
LIN {X 0,Y 193.247,Z 245.399,A -85,B 0,C 180,E1 -21957.916,E2 -21957.916} C_VEL
LIN {X 0,Y 193.422,Z 245.387,A -85,B 0,C 180,E1 -21960,E2 -21960} C_VEL
LIN {X 0,Y 192.932,Z 245.442,A -85,B 0,C 180,E1 -21964.178,E2 -21964.178} C_VEL
LIN {X 0,Y 193.009,Z 245.429,A -85,B 0,C 180,E1 -21968.375,E2 -21968.375} C_VEL
LIN {X 0,Y 192.779,Z 245.456,A -85,B 0,C 180,E1 -21972.635,E2 -21972.635} C_VEL
LIN {X 0,Y 192.705,Z 245.467,A -85,B 0,C 180,E1 -21976.963,E2 -21976.963} C_VEL
LIN {X 0,Y 192.571,Z 245.484,A -85,B 0,C 180,E1 -21981.405,E2 -21981.405} C_VEL
LIN {X 0,Y 192.612,Z 245.488,A -85,B 0,C 180,E1 -21984.192,E2 -21984.192} C_VEL
LIN {X 0,Y 192.546,Z 245.489,A -85,B 0,C 180,E1 -21989.625,E2 -21989.625} C_VEL
LIN {X 0,Y 194.24,Z 250.361,A -85,B 0,C 180,E1 -21994.19,E2 -21994.19} C_VEL
LIN {X 0,Y 197.94,Z 255.786,A -85,B 0,C 180,E1 -21996.409,E2 -21996.409} C_VEL
LIN {X 0,Y 199.29,Z 257.551,A -85,B 0,C 180,E1 -21997.151,E2 -21997.151} C_VEL
LIN {X 0,Y 202.693,Z 262.469,A -85,B 0,C 180,E1 -21998.936,E2 -21998.936} C_VEL
LIN {X 0,Y 207.792,Z 270.609,A -85,B 0,C 180,E1 -22001.408,E2 -22001.408} C_VEL
LIN {X 0,Y 211.014,Z 275.939,A -85,B 0,C 180,E1 -22002.852,E2 -22002.852} C_VEL
LIN {X 0,Y 215.861,Z 284.421,A -85,B 0,C 180,E1 -22004.886,E2 -22004.886} C_VEL
LIN {X 0,Y 221.785,Z 296.1,A -85,B 0,C 180,E1 -22007.205,E2 -22007.205} C_VEL
